LIN {X -0.049,Y -582.708,Z 976.726,A 0.000,B 0.000,C 90.000,E1 346.756} C_DIS
LIN {X 0.095,Y -587.097,Z 976.722,A 0.000,B 0.000,C 90.000,E1 345.936} C_DIS
LIN {X -0.292,Y -591.184,Z 976.718,A 0.000,B 0.000,C 90.000,E1 345.172} C_DIS
LIN {X -0.216,Y -596.425,Z 976.712,A 0.000,B 0.000,C 90.000,E1 344.102} C_DIS
LIN {X 0.105,Y -601.361,Z 976.706,A 0.000,B 0.000,C 90.000,E1 343.015} C_DIS
LIN {X 0.020,Y -604.929,Z 976.701,A 0.000,B 0.000,C 90.000,E1 342.236} C_DIS
LIN {X 0.200,Y -610.324,Z 976.694,A 0.000,B 0.000,C 90.000,E1 340.913} C_DIS
LIN {X 0.140,Y -614.377,Z 976.688,A 0.000,B 0.000,C 90.000,E1 339.880} C_DIS
LIN {X 0.129,Y -618.154,Z 976.683,A 0.000,B 0.000,C 90.000,E1 338.847} C_DIS
LIN {X -0.183,Y -621.682,Z 976.677,A 0.000,B 0.000,C 90.000,E1 337.847} C_DIS
LIN {X 0.136,Y -625.716,Z 976.670,A 0.000,B 0.000,C 90.000,E1 336.538} C_DIS
LIN {X -0.067,Y -628.774,Z 976.664,A 0.000,B 0.000,C 90.000,E1 335.537} C_DIS
LIN {X -0.237,Y -631.659,Z 976.658,A 0.000,B 0.000,C 90.000,E1 334.537} C_DIS
LIN {X -0.099,Y -634.157,Z 976.653,A 0.000,B 0.000,C 90.000,E1 333.512} C_DIS
LIN {X 0.073,Y -636.573,Z 976.647,A 0.000,B 0.000,C 90.000,E1 332.487} C_DIS
LIN {X 0.129,Y -639.825,Z 976.639,A 0.000,B 0.000,C 90.000,E1 330.973} C_DIS
LIN {X -0.192,Y -641.817,Z 976.633,A 0.000,B 0.000,C 90.000,E1 329.999} C_DIS
LIN {X -0.169,Y -643.706,Z 976.628,A 0.000,B 0.000,C 90.000,E1 328.997} C_DIS
LIN {X -0.122,Y -645.317,Z 976.622,A 0.000,B 0.000,C 90.000,E1 327.995} C_DIS
LIN {X -0.061,Y -646.790,Z 976.617,A 0.000,B 0.000,C 90.000,E1 326.993} C_DIS
LIN {X -0.107,Y -648.333,Z 976.610,A 0.000,B 0.000,C 90.000,E1 325.754} C_DIS
LIN {X -0.191,Y -649.344,Z 976.604,A 0.000,B 0.000,C 90.000,E1 324.769} C_DIS
LIN {X 0.098,Y -650.530,Z 976.596,A 0.000,B 0.000,C 90.000,E1 323.256} C_DIS
LIN {X 0.014,Y -651.473,Z 976.588,A 0.000,B 0.000,C 90.000,E1 321.778} C_DIS
LIN {X -0.206,Y -652.064,Z 976.581,A 0.000,B 0.000,C 90.000,E1 320.561} C_DIS
LIN {X 0.057,Y -652.847,Z 976.571,A 0.000,B 0.000,C 90.000,E1 318.809} C_DIS
LIN {X -0.360,Y -654.469,Z 976.558,A 0.000,B 0.000,C 90.000,E1 316.377} C_DIS
LIN {X -0.086,Y -655.453,Z 976.551,A 0.000,B 0.000,C 90.000,E1 315.121} C_DIS
LIN {X 0.068,Y -657.207,Z 976.538,A 0.000,B 0.000,C 90.000,E1 312.894} C_DIS
LIN {X -0.085,Y -658.420,Z 976.530,A 0.000,B 0.000,C 90.000,E1 311.434} C_DIS
LIN {X 0.317,Y -659.253,Z 976.523,A 0.000,B 0.000,C 90.000,E1 310.172} C_DIS
LIN {X -0.186,Y -660.046,Z 976.517,A 0.000,B 0.000,C 90.000,E1 308.991} C_DIS
LIN {X -0.199,Y -660.753,Z 976.508,A 0.000,B 0.000,C 90.000,E1 307.523} C_DIS
LIN {X -0.205,Y -661.096,Z 976.504,A 0.000,B 0.000,C 90.000,E1 306.790} C_DIS
LIN {X 0.408,Y -661.427,Z 976.495,A 0.000,B 0.000,C 90.000,E1 305.025} C_DIS
LIN {X -0.267,Y -661.847,Z 976.485,A 0.000,B 0.000,C 90.000,E1 303.372} C_DIS
LIN {X 0.062,Y -663.392,Z 976.469,A 0.000,B 0.000,C 90.000,E1 300.413} C_DIS
LIN {X 0.159,Y -669.765,Z 976.442,A 0.000,B 0.000,C 90.000,E1 295.540} C_DIS
LIN {X 0.099,Y -671.892,Z 976.435,A 0.000,B 0.000,C 90.000,E1 294.335} C_DIS
LIN {X -0.109,Y -673.447,Z 976.430,A 0.000,B 0.000,C 90.000,E1 293.387} C_DIS
LIN {X -0.030,Y -674.165,Z 976.427,A 0.000,B 0.000,C 90.000,E1 292.898} C_DIS
LIN {X 0.058,Y -674.564,Z 976.425,A 0.000,B 0.000,C 90.000,E1 292.408} C_DIS
LIN {X 0.231,Y -674.612,Z 976.423,A 0.000,B 0.000,C 90.000,E1 292.153} C_DIS
LIN {X -0.302,Y -674.336,Z 976.421,A 0.000,B 0.000,C 90.000,E1 291.716} C_DIS
LIN {X -0.133,Y -673.871,Z 976.419,A 0.000,B 0.000,C 90.000,E1 291.461} C_DIS
LIN {X -0.210,Y -673.270,Z 976.418,A 0.000,B 0.000,C 90.000,E1 291.227} C_DIS
LIN {X -0.044,Y -672.447,Z 976.417,A 0.000,B 0.000,C 90.000,E1 290.972} C_DIS
LIN {X 0.036,Y -671.818,Z 976.416,A 0.000,B 0.000,C 90.000,E1 290.844} C_DIS
LIN {X -0.121,Y -670.864,Z 976.415,A 0.000,B 0.000,C 90.000,E1 290.737} C_DIS
LIN {X 0.152,Y -665.304,Z 976.412,A 0.000,B 0.000,C 90.000,E1 290.194} C_DIS
LIN {X -0.021,Y -657.463,Z 976.409,A 0.000,B 0.000,C 90.000,E1 289.704} C_DIS
LIN {X -0.276,Y -653.001,Z 976.408,A 0.000,B 0.000,C 90.000,E1 289.450} C_DIS
LIN {X 0.214,Y -651.160,Z 976.407,A 0.000,B 0.000,C 90.000,E1 289.214} C_DIS
LIN {X 0.171,Y -651.142,Z 976.407,A 0.000,B 0.000,C 90.000,E1 289.214} C_DIS
LIN {X 0.129,Y -651.087,Z 976.406,A 0.000,B 0.000,C 90.000,E1 289.141} C_DIS
LIN {X -0.058,Y -652.540,Z 976.404,A 0.000,B 0.000,C 90.000,E1 288.725} C_DIS
LIN {X -0.127,Y -656.444,Z 976.400,A 0.000,B 0.000,C 90.000,E1 288.055} C_DIS
LIN {X -0.091,Y -660.813,Z 976.396,A 0.000,B 0.000,C 90.000,E1 287.330} C_DIS
LIN {X -0.246,Y -664.149,Z 976.393,A 0.000,B 0.000,C 90.000,E1 286.732} C_DIS
LIN {X 0.317,Y -667.054,Z 976.390,A 0.000,B 0.000,C 90.000,E1 286.079} C_DIS
LIN {X 0.081,Y -669.685,Z 976.385,A 0.000,B 0.000,C 90.000,E1 285.371} C_DIS
LIN {X -0.060,Y -671.033,Z 976.383,A 0.000,B 0.000,C 90.000,E1 284.898} C_DIS
LIN {X -0.087,Y -672.571,Z 976.379,A 0.000,B 0.000,C 90.000,E1 284.175} C_DIS
LIN {X 0.383,Y -673.703,Z 976.375,A 0.000,B 0.000,C 90.000,E1 283.411} C_DIS
LIN {X 0.060,Y -674.413,Z 976.371,A 0.000,B 0.000,C 90.000,E1 282.715} C_DIS
LIN {X -0.103,Y -674.841,Z 976.367,A 0.000,B 0.000,C 90.000,E1 282.007} C_DIS
LIN {X -0.271,Y -674.764,Z 976.363,A 0.000,B 0.000,C 90.000,E1 281.299} C_DIS
LIN {X 0.148,Y -674.517,Z 976.360,A 0.000,B 0.000,C 90.000,E1 280.782} C_DIS
LIN {X 0.031,Y -673.995,Z 976.357,A 0.000,B 0.000,C 90.000,E1 280.310} C_DIS
LIN {X -0.210,Y -673.266,Z 976.355,A 0.000,B 0.000,C 90.000,E1 279.849} C_DIS
LIN {X 0.322,Y -672.220,Z 976.352,A 0.000,B 0.000,C 90.000,E1 279.321} C_DIS
LIN {X 0.075,Y -670.878,Z 976.349,A 0.000,B 0.000,C 90.000,E1 278.859} C_DIS
LIN {X -0.001,Y -670.147,Z 976.348,A 0.000,B 0.000,C 90.000,E1 278.624} C_DIS
LIN {X -0.259,Y -668.440,Z 976.345,A 0.000,B 0.000,C 90.000,E1 278.163} C_DIS
LIN {X 0.136,Y -666.393,Z 976.343,A 0.000,B 0.000,C 90.000,E1 277.644} C_DIS
LIN {X -0.234,Y -663.311,Z 976.339,A 0.000,B 0.000,C 90.000,E1 277.068} C_DIS
LIN {X 0.104,Y -659.603,Z 976.336,A 0.000,B 0.000,C 90.000,E1 276.429} C_DIS
LIN {X 0.330,Y -655.150,Z 976.332,A 0.000,B 0.000,C 90.000,E1 275.796} C_DIS
LIN {X -0.022,Y -651.196,Z 976.330,A 0.000,B 0.000,C 90.000,E1 275.334} C_DIS
LIN {X 0.191,Y -646.922,Z 976.327,A 0.000,B 0.000,C 90.000,E1 274.821} C_DIS
LIN {X -0.211,Y -642.262,Z 976.324,A 0.000,B 0.000,C 90.000,E1 274.359} C_DIS
LIN {X 0.043,Y -635.920,Z 976.321,A 0.000,B 0.000,C 90.000,E1 273.726} C_DIS
LIN {X -0.093,Y -630.643,Z 976.318,A 0.000,B 0.000,C 90.000,E1 273.269} C_DIS
LIN {X 0.021,Y -625.023,Z 976.316,A 0.000,B 0.000,C 90.000,E1 272.808} C_DIS
LIN {X -0.203,Y -617.622,Z 976.313,A 0.000,B 0.000,C 90.000,E1 272.293} C_DIS
LIN {X -0.222,Y -611.469,Z 976.310,A 0.000,B 0.000,C 90.000,E1 271.892} C_DIS
LIN {X -0.230,Y -603.376,Z 976.308,A 0.000,B 0.000,C 90.000,E1 271.432} C_DIS
LIN {X 0.110,Y -598.334,Z 976.306,A 0.000,B 0.000,C 90.000,E1 271.146} C_DIS
LIN {X -0.088,Y -591.281,Z 976.305,A 0.000,B 0.000,C 90.000,E1 270.859} C_DIS
LIN {X 0.063,Y -584.127,Z 976.303,A 0.000,B 0.000,C 90.000,E1 270.573} C_DIS
LIN {X 0.103,Y -576.473,Z 976.302,A 0.000,B 0.000,C 90.000,E1 270.344} C_DIS
LIN {X -0.244,Y -571.044,Z 976.301,A 0.000,B 0.000,C 90.000,E1 270.229} C_DIS
LIN {X 0.130,Y -564.562,Z 976.300,A 0.000,B 0.000,C 90.000,E1 270.057} C_DIS
LIN {X 0.026,Y -557.390,Z 976.300,A 0.000,B 0.000,C 90.000,E1 270.000} C_DIS
LIN {X -0.024,Y -546.296,Z 976.300,A 0.000,B 0.000,C 90.000,E1 270.000} C_DIS
LIN {X -0.220,Y -544.017,Z 976.300,A 0.000,B 0.000,C 90.000,E1 269.943} C_DIS
LIN {X 0.151,Y -543.248,Z 976.299,A 0.000,B 0.000,C 90.000,E1 269.885} C_DIS
LIN {X 0.108,Y -543.043,Z 976.299,A 0.000,B 0.000,C 90.000,E1 269.885} C_DIS
LIN {X -0.079,Y -542.595,Z 976.298,A 0.000,B 0.000,C 90.000,E1 269.714} C_DIS
LIN {X -0.251,Y -541.922,Z 976.293,A 0.000,B 0.000,C 90.000,E1 268.740} C_DIS
LIN {X -0.045,Y -540.496,Z 976.282,A 0.000,B 0.000,C 90.000,E1 266.731} C_DIS
LIN {X 0.063,Y -539.552,Z 976.274,A 0.000,B 0.000,C 90.000,E1 265.298} C_DIS
LIN {X 0.240,Y -538.503,Z 976.266,A 0.000,B 0.000,C 90.000,E1 263.856} C_DIS
LIN {X -0.127,Y -537.229,Z 976.258,A 0.000,B 0.000,C 90.000,E1 262.470} C_DIS
LIN {X -0.048,Y -536.080,Z 976.252,A 0.000,B 0.000,C 90.000,E1 261.319} C_DIS
LIN {X 0.230,Y -534.668,Z 976.244,A 0.000,B 0.000,C 90.000,E1 259.859} C_DIS
LIN {X -0.087,Y -532.682,Z 976.234,A 0.000,B 0.000,C 90.000,E1 258.173} C_DIS
LIN {X 0.046,Y -531.778,Z 976.229,A 0.000,B 0.000,C 90.000,E1 257.297} C_DIS
LIN {X 0.041,Y -529.264,Z 976.218,A 0.000,B 0.000,C 90.000,E1 255.283} C_DIS
LIN {X -0.204,Y -527.751,Z 976.210,A 0.000,B 0.000,C 90.000,E1 253.866} C_DIS
LIN {X -0.176,Y -525.901,Z 976.201,A 0.000,B 0.000,C 90.000,E1 252.127} C_DIS
LIN {X -0.186,Y -524.098,Z 976.193,A 0.000,B 0.000,C 90.000,E1 250.678} C_DIS
LIN {X 0.102,Y -521.788,Z 976.183,A 0.000,B 0.000,C 90.000,E1 248.901} C_DIS
LIN {X -0.295,Y -519.948,Z 976.175,A 0.000,B 0.000,C 90.000,E1 247.486} C_DIS
LIN {X -0.001,Y -519.209,Z 976.172,A 0.000,B 0.000,C 90.000,E1 246.869} C_DIS
LIN {X 0.099,Y -516.564,Z 976.162,A 0.000,B 0.000,C 90.000,E1 245.101} C_DIS
LIN {X 0.023,Y -514.257,Z 976.154,A 0.000,B 0.000,C 90.000,E1 243.640} C_DIS
LIN {X -0.208,Y -512.415,Z 976.147,A 0.000,B 0.000,C 90.000,E1 242.487} C_DIS
LIN {X 0.112,Y -510.012,Z 976.139,A 0.000,B 0.000,C 90.000,E1 240.973} C_DIS
LIN {X -0.306,Y -507.426,Z 976.131,A 0.000,B 0.000,C 90.000,E1 239.537} C_DIS
LIN {X -0.142,Y -505.116,Z 976.124,A 0.000,B 0.000,C 90.000,E1 238.329} C_DIS
LIN {X -0.134,Y -502.056,Z 976.116,A 0.000,B 0.000,C 90.000,E1 236.834} C_DIS
LIN {X 0.218,Y -499.376,Z 976.109,A 0.000,B 0.000,C 90.000,E1 235.595} C_DIS
LIN {X -0.151,Y -495.265,Z 976.099,A 0.000,B 0.000,C 90.000,E1 233.829} C_DIS
LIN {X 0.227,Y -491.712,Z 976.091,A 0.000,B 0.000,C 90.000,E1 232.271} C_DIS
LIN {X -0.083,Y -488.934,Z 976.084,A 0.000,B 0.000,C 90.000,E1 231.090} C_DIS
LIN {X -0.094,Y -484.579,Z 976.074,A 0.000,B 0.000,C 90.000,E1 229.256} C_DIS
LIN {X 0.057,Y -480.376,Z 976.063,A 0.000,B 0.000,C 90.000,E1 227.391} C_DIS
LIN {X -0.228,Y -476.328,Z 976.053,A 0.000,B 0.000,C 90.000,E1 225.567} C_DIS
LIN {X 0.300,Y -472.927,Z 976.044,A 0.000,B 0.000,C 90.000,E1 223.947} C_DIS
LIN {X 0.192,Y -468.772,Z 976.034,A 0.000,B 0.000,C 90.000,E1 222.081} C_DIS
LIN {X 0.102,Y -466.768,Z 976.029,A 0.000,B 0.000,C 90.000,E1 221.148} C_DIS
LIN {X 0.146,Y -463.236,Z 976.020,A 0.000,B 0.000,C 90.000,E1 219.564} C_DIS
LIN {X -0.049,Y -458.183,Z 976.008,A 0.000,B 0.000,C 90.000,E1 217.363} C_DIS
LIN {X -0.017,Y -453.957,Z 975.997,A 0.000,B 0.000,C 90.000,E1 215.438} C_DIS
LIN {X 0.026,Y -449.715,Z 975.986,A 0.000,B 0.000,C 90.000,E1 213.499} C_DIS
LIN {X 0.035,Y -446.193,Z 975.977,A 0.000,B 0.000,C 90.000,E1 211.878} C_DIS
LIN {X -0.084,Y -443.427,Z 975.970,A 0.000,B 0.000,C 90.000,E1 210.590} C_DIS
LIN {X -0.088,Y -440.629,Z 975.963,A 0.000,B 0.000,C 90.000,E1 209.283} C_DIS
LIN {X 0.139,Y -435.508,Z 975.950,A 0.000,B 0.000,C 90.000,E1 206.950} C_DIS
LIN {X -0.005,Y -433.380,Z 975.944,A 0.000,B 0.000,C 90.000,E1 205.976} C_DIS
LIN {X 0.023,Y -430.297,Z 975.937,A 0.000,B 0.000,C 90.000,E1 204.643} C_DIS
LIN {X -0.074,Y -423.467,Z 975.920,A 0.000,B 0.000,C 90.000,E1 201.642} C_DIS
LIN {X -0.023,Y -418.394,Z 975.907,A 0.000,B 0.000,C 90.000,E1 199.268} C_DIS
LIN {X -0.100,Y -413.003,Z 975.892,A 0.000,B 0.000,C 90.000,E1 196.551} C_DIS
LIN {X -0.036,Y -409.182,Z 975.880,A 0.000,B 0.000,C 90.000,E1 194.481} C_DIS
LIN {X -0.163,Y -405.944,Z 975.871,A 0.000,B 0.000,C 90.000,E1 192.771} C_DIS
LIN {X 0.034,Y -402.616,Z 975.861,A 0.000,B 0.000,C 90.000,E1 191.007} C_DIS
LIN {X 0.014,Y -400.007,Z 975.853,A 0.000,B 0.000,C 90.000,E1 189.613} C_DIS
LIN {X 0.032,Y -393.198,Z 975.832,A 0.000,B 0.000,C 90.000,E1 185.739} C_DIS
LIN {X -0.146,Y -392.071,Z 975.826,A 0.000,B 0.000,C 90.000,E1 184.702} C_DIS
LIN {X 0.105,Y -391.526,Z 975.822,A 0.000,B 0.000,C 90.000,E1 183.955} C_DIS
LIN {X 0.021,Y -391.404,Z 975.820,A 0.000,B 0.000,C 90.000,E1 183.612} C_DIS
LIN {X -0.124,Y -391.727,Z 975.816,A 0.000,B 0.000,C 90.000,E1 182.922} C_DIS
LIN {X 0.185,Y -392.168,Z 975.814,A 0.000,B 0.000,C 90.000,E1 182.522} C_DIS
LIN {X 0.105,Y -392.821,Z 975.812,A 0.000,B 0.000,C 90.000,E1 182.178} C_DIS
LIN {X 0.115,Y -393.673,Z 975.810,A 0.000,B 0.000,C 90.000,E1 181.835} C_DIS
LIN {X 0.047,Y -395.519,Z 975.807,A 0.000,B 0.000,C 90.000,E1 181.318} C_DIS
LIN {X 0.012,Y -397.225,Z 975.805,A 0.000,B 0.000,C 90.000,E1 180.974} C_DIS
LIN {X -0.050,Y -399.256,Z 975.804,A 0.000,B 0.000,C 90.000,E1 180.630} C_DIS
LIN {X -0.136,Y -402.294,Z 975.801,A 0.000,B 0.000,C 90.000,E1 180.229} C_DIS
LIN {X -0.169,Y -405.098,Z 975.799,A 0.000,B 0.000,C 90.000,E1 179.885} C_DIS
LIN {X -0.073,Y -412.702,Z 975.795,A 0.000,B 0.000,C 90.000,E1 179.083} C_DIS
LIN {X 0.071,Y -424.664,Z 975.789,A 0.000,B 0.000,C 90.000,E1 177.936} C_DIS
LIN {X 0.118,Y -436.561,Z 975.782,A 0.000,B 0.000,C 90.000,E1 176.788} C_DIS
LIN {X -0.066,Y -440.929,Z 975.780,A 0.000,B 0.000,C 90.000,E1 176.388} C_DIS
LIN {X -0.137,Y -449.606,Z 975.775,A 0.000,B 0.000,C 90.000,E1 175.527} C_DIS
LIN {X 0.185,Y -460.939,Z 975.769,A 0.000,B 0.000,C 90.000,E1 174.318} C_DIS
LIN {X 0.115,Y -470.380,Z 975.763,A 0.000,B 0.000,C 90.000,E1 173.280} C_DIS
LIN {X 0.092,Y -478.131,Z 975.758,A 0.000,B 0.000,C 90.000,E1 172.356} C_DIS
LIN {X 0.048,Y -485.586,Z 975.753,A 0.000,B 0.000,C 90.000,E1 171.432} C_DIS
LIN {X 0.059,Y -494.990,Z 975.746,A 0.000,B 0.000,C 90.000,E1 170.208} C_DIS
LIN {X -0.040,Y -502.686,Z 975.740,A 0.000,B 0.000,C 90.000,E1 169.162} C_DIS
LIN {X 0.231,Y -510.899,Z 975.733,A 0.000,B 0.000,C 90.000,E1 167.937} C_DIS
LIN {X 0.250,Y -520.550,Z 975.725,A 0.000,B 0.000,C 90.000,E1 166.464} C_DIS
LIN {X 0.063,Y -524.967,Z 975.721,A 0.000,B 0.000,C 90.000,E1 165.755} C_DIS
LIN {X -0.066,Y -531.342,Z 975.715,A 0.000,B 0.000,C 90.000,E1 164.755} C_DIS
LIN {X -0.133,Y -538.234,Z 975.709,A 0.000,B 0.000,C 90.000,E1 163.614} C_DIS
LIN {X -0.257,Y -544.932,Z 975.703,A 0.000,B 0.000,C 90.000,E1 162.489} C_DIS
LIN {X 0.134,Y -553.029,Z 975.695,A 0.000,B 0.000,C 90.000,E1 161.040} C_DIS
LIN {X -0.068,Y -560.210,Z 975.688,A 0.000,B 0.000,C 90.000,E1 159.806} C_DIS
LIN {X 0.150,Y -564.674,Z 975.683,A 0.000,B 0.000,C 90.000,E1 158.954} C_DIS
LIN {X 0.229,Y -570.421,Z 975.677,A 0.000,B 0.000,C 90.000,E1 157.847} C_DIS
LIN {X 0.019,Y -574.548,Z 975.673,A 0.000,B 0.000,C 90.000,E1 157.050} C_DIS
LIN {X 0.149,Y -577.818,Z 975.669,A 0.000,B 0.000,C 90.000,E1 156.357} C_DIS
LIN {X 0.175,Y -582.234,Z 975.664,A 0.000,B 0.000,C 90.000,E1 155.409} C_DIS
LIN {X 0.253,Y -586.241,Z 975.658,A 0.000,B 0.000,C 90.000,E1 154.460} C_DIS
LIN {X -0.099,Y -589.497,Z 975.654,A 0.000,B 0.000,C 90.000,E1 153.691} C_DIS
LIN {X 0.007,Y -593.406,Z 975.648,A 0.000,B 0.000,C 90.000,E1 152.615} C_DIS
LIN {X -0.088,Y -596.866,Z 975.642,A 0.000,B 0.000,C 90.000,E1 151.563} C_DIS
LIN {X -0.208,Y -600.991,Z 975.635,A 0.000,B 0.000,C 90.000,E1 150.255} C_DIS
LIN {X 0.044,Y -605.049,Z 975.627,A 0.000,B 0.000,C 90.000,E1 148.918} C_DIS
LIN {X 0.104,Y -608.260,Z 975.622,A 0.000,B 0.000,C 90.000,E1 147.867} C_DIS
LIN {X 0.012,Y -611.516,Z 975.616,A 0.000,B 0.000,C 90.000,E1 146.834} C_DIS
LIN {X 0.009,Y -617.095,Z 975.606,A 0.000,B 0.000,C 90.000,E1 145.022} C_DIS
LIN {X -0.192,Y -621.794,Z 975.597,A 0.000,B 0.000,C 90.000,E1 143.497} C_DIS
LIN {X -0.056,Y -626.495,Z 975.589,A 0.000,B 0.000,C 90.000,E1 141.949} C_DIS
LIN {X -0.209,Y -631.159,Z 975.580,A 0.000,B 0.000,C 90.000,E1 140.436} C_DIS
LIN {X -0.367,Y -635.644,Z 975.572,A 0.000,B 0.000,C 90.000,E1 138.933} C_DIS
LIN {X 0.195,Y -642.570,Z 975.559,A 0.000,B 0.000,C 90.000,E1 136.620} C_DIS
LIN {X -0.247,Y -647.308,Z 975.551,A 0.000,B 0.000,C 90.000,E1 135.162} C_DIS
LIN {X -0.304,Y -655.718,Z 975.537,A 0.000,B 0.000,C 90.000,E1 132.690} C_DIS
LIN {X -0.057,Y -664.670,Z 975.523,A 0.000,B 0.000,C 90.000,E1 130.216} C_DIS
LIN {X -0.041,Y -668.186,Z 975.518,A 0.000,B 0.000,C 90.000,E1 129.241} C_DIS
LIN {X -0.299,Y -673.284,Z 975.510,A 0.000,B 0.000,C 90.000,E1 127.810} C_DIS
LIN {X -0.047,Y -677.105,Z 975.503,A 0.000,B 0.000,C 90.000,E1 126.583} C_DIS
LIN {X -0.133,Y -680.780,Z 975.497,A 0.000,B 0.000,C 90.000,E1 125.391} C_DIS
LIN {X 0.222,Y -683.642,Z 975.491,A 0.000,B 0.000,C 90.000,E1 124.405} C_DIS
LIN {X -0.143,Y -686.979,Z 975.485,A 0.000,B 0.000,C 90.000,E1 123.245} C_DIS
LIN {X 0.131,Y -690.701,Z 975.477,A 0.000,B 0.000,C 90.000,E1 121.799} C_DIS
LIN {X -0.134,Y -693.018,Z 975.471,A 0.000,B 0.000,C 90.000,E1 120.875} C_DIS
LIN {X 0.340,Y -694.597,Z 975.468,A 0.000,B 0.000,C 90.000,E1 120.129} C_DIS
LIN {X -0.126,Y -695.992,Z 975.464,A 0.000,B 0.000,C 90.000,E1 119.461} C_DIS
LIN {X 0.283,Y -697.433,Z 975.458,A 0.000,B 0.000,C 90.000,E1 118.487} C_DIS
LIN {X 0.037,Y -698.610,Z 975.452,A 0.000,B 0.000,C 90.000,E1 117.334} C_DIS
LIN {X 0.215,Y -699.315,Z 975.448,A 0.000,B 0.000,C 90.000,E1 116.616} C_DIS
LIN {X -0.003,Y -700.165,Z 975.442,A 0.000,B 0.000,C 90.000,E1 115.463} C_DIS
LIN {X -0.122,Y -700.448,Z 975.438,A 0.000,B 0.000,C 90.000,E1 114.771} C_DIS
LIN {X 0.130,Y -700.507,Z 975.435,A 0.000,B 0.000,C 90.000,E1 114.283} C_DIS
LIN {X 0.032,Y -700.124,Z 975.432,A 0.000,B 0.000,C 90.000,E1 113.823} C_DIS
LIN {X 0.019,Y -699.837,Z 975.431,A 0.000,B 0.000,C 90.000,E1 113.590} C_DIS
LIN {X -0.090,Y -698.362,Z 975.429,A 0.000,B 0.000,C 90.000,E1 113.131} C_DIS
LIN {X -0.101,Y -697.334,Z 975.427,A 0.000,B 0.000,C 90.000,E1 112.898} C_DIS
LIN {X 0.156,Y -695.329,Z 975.426,A 0.000,B 0.000,C 90.000,E1 112.642} C_DIS
LIN {X 0.262,Y -691.942,Z 975.424,A 0.000,B 0.000,C 90.000,E1 112.280} C_DIS
LIN {X -0.257,Y -690.182,Z 975.423,A 0.000,B 0.000,C 90.000,E1 112.206} C_DIS
LIN {X 0.245,Y -685.451,Z 975.422,A 0.000,B 0.000,C 90.000,E1 111.972} C_DIS
LIN {X 0.347,Y -683.290,Z 975.422,A 0.000,B 0.000,C 90.000,E1 111.897} C_DIS
LIN {X -0.209,Y -675.865,Z 975.421,A 0.000,B 0.000,C 90.000,E1 111.770} C_DIS
LIN {X 0.240,Y -674.512,Z 975.421,A 0.000,B 0.000,C 90.000,E1 111.716} C_DIS
LIN {X 0.175,Y -672.657,Z 975.421,A 0.000,B 0.000,C 90.000,E1 111.716} C_DIS
LIN {X 0.104,Y -626.026,Z 975.421,A 0.000,B 0.000,C 90.000,E1 111.716} C_DIS
LIN {X -0.147,Y -621.534,Z 975.420,A 0.000,B 0.000,C 90.000,E1 111.663} C_DIS
LIN {X -0.200,Y -615.743,Z 975.420,A 0.000,B 0.000,C 90.000,E1 111.535} C_DIS
LIN {X -0.047,Y -610.298,Z 975.419,A 0.000,B 0.000,C 90.000,E1 111.354} C_DIS
LIN {X -0.253,Y -603.607,Z 975.417,A 0.000,B 0.000,C 90.000,E1 111.099} C_DIS
LIN {X 0.138,Y -597.489,Z 975.415,A 0.000,B 0.000,C 90.000,E1 110.737} C_DIS
LIN {X -0.152,Y -590.496,Z 975.413,A 0.000,B 0.000,C 90.000,E1 110.301} C_DIS
LIN {X 0.287,Y -578.355,Z 975.408,A 0.000,B 0.000,C 90.000,E1 109.322} C_DIS
LIN {X -0.163,Y -573.848,Z 975.406,A 0.000,B 0.000,C 90.000,E1 109.033} C_DIS
LIN {X 0.152,Y -567.242,Z 975.403,A 0.000,B 0.000,C 90.000,E1 108.598} C_DIS
LIN {X 0.208,Y -552.115,Z 975.399,A 0.000,B 0.000,C 90.000,E1 107.819} C_DIS
LIN {X 0.101,Y -549.945,Z 975.398,A 0.000,B 0.000,C 90.000,E1 107.638} C_DIS
LIN {X 0.064,Y -549.916,Z 975.398,A 0.000,B 0.000,C 90.000,E1 107.638} C_DIS
LIN {X -0.275,Y -549.445,Z 975.397,A 0.000,B 0.000,C 90.000,E1 107.402} C_DIS
LIN {X -0.059,Y -549.569,Z 975.393,A 0.000,B 0.000,C 90.000,E1 106.677} C_DIS
LIN {X -0.107,Y -550.406,Z 975.382,A 0.000,B 0.000,C 90.000,E1 104.717} C_DIS
LIN {X -0.266,Y -551.503,Z 975.371,A 0.000,B 0.000,C 90.000,E1 102.771} C_DIS
LIN {X -0.152,Y -553.940,Z 975.355,A 0.000,B 0.000,C 90.000,E1 99.962} C_DIS
LIN {X -0.041,Y -555.670,Z 975.346,A 0.000,B 0.000,C 90.000,E1 98.276} C_DIS
LIN {X -0.046,Y -557.231,Z 975.337,A 0.000,B 0.000,C 90.000,E1 96.606} C_DIS
LIN {X -0.083,Y -558.317,Z 975.329,A 0.000,B 0.000,C 90.000,E1 95.220} C_DIS
LIN {X -0.160,Y -559.230,Z 975.321,A 0.000,B 0.000,C 90.000,E1 93.841} C_DIS
LIN {X 0.126,Y -559.732,Z 975.317,A 0.000,B 0.000,C 90.000,E1 92.980} C_DIS
LIN {X 0.037,Y -560.476,Z 975.309,A 0.000,B 0.000,C 90.000,E1 91.604} C_DIS
LIN {X 0.045,Y -561.266,Z 975.300,A 0.000,B 0.000,C 90.000,E1 89.943} C_DIS
LIN {X -0.028,Y -561.686,Z 975.292,A 0.000,B 0.000,C 90.000,E1 88.568} C_DIS
LIN {X 0.012,Y -562.097,Z 975.283,A 0.000,B 0.000,C 90.000,E1 86.906} C_DIS
LIN {X -0.004,Y -562.312,Z 975.275,A 0.000,B 0.000,C 90.000,E1 85.527} C_DIS
LIN {X 0.219,Y -562.559,Z 975.264,A 0.000,B 0.000,C 90.000,E1 83.571} C_DIS
LIN {X 0.096,Y -562.955,Z 975.252,A 0.000,B 0.000,C 90.000,E1 81.376} C_DIS
LIN {X 0.004,Y -563.655,Z 975.241,A 0.000,B 0.000,C 90.000,E1 79.454} C_DIS
LIN {X 0.215,Y -564.684,Z 975.229,A 0.000,B 0.000,C 90.000,E1 77.229} C_DIS
LIN {X 0.031,Y -566.117,Z 975.217,A 0.000,B 0.000,C 90.000,E1 75.046} C_DIS
LIN {X -0.142,Y -567.444,Z 975.206,A 0.000,B 0.000,C 90.000,E1 73.142} C_DIS
LIN {X -0.081,Y -568.345,Z 975.199,A 0.000,B 0.000,C 90.000,E1 71.764} C_DIS
LIN {X -0.019,Y -569.347,Z 975.190,A 0.000,B 0.000,C 90.000,E1 70.115} C_DIS
LIN {X 0.253,Y -570.077,Z 975.182,A 0.000,B 0.000,C 90.000,E1 68.720} C_DIS
LIN {X -0.147,Y -570.536,Z 975.176,A 0.000,B 0.000,C 90.000,E1 67.667} C_DIS
LIN {X -0.188,Y -571.056,Z 975.168,A 0.000,B 0.000,C 90.000,E1 66.305} C_DIS
LIN {X -0.164,Y -571.570,Z 975.159,A 0.000,B 0.000,C 90.000,E1 64.665} C_DIS
LIN {X 0.287,Y -571.934,Z 975.152,A 0.000,B 0.000,C 90.000,E1 63.256} C_DIS
LIN {X 0.237,Y -572.190,Z 975.144,A 0.000,B 0.000,C 90.000,E1 61.897} C_DIS
LIN {X 0.020,Y -572.367,Z 975.135,A 0.000,B 0.000,C 90.000,E1 60.284} C_DIS
LIN {X -0.125,Y -572.538,Z 975.126,A 0.000,B 0.000,C 90.000,E1 58.663} C_DIS
LIN {X -0.255,Y -572.717,Z 975.117,A 0.000,B 0.000,C 90.000,E1 57.041} C_DIS
LIN {X -0.210,Y -572.707,Z 975.109,A 0.000,B 0.000,C 90.000,E1 55.674} C_DIS
LIN {X -0.123,Y -572.624,Z 975.105,A 0.000,B 0.000,C 90.000,E1 54.848} C_DIS
LIN {X -0.030,Y -572.276,Z 975.099,A 0.000,B 0.000,C 90.000,E1 53.749} C_DIS
LIN {X 0.047,Y -571.928,Z 975.094,A 0.000,B 0.000,C 90.000,E1 52.924} C_DIS
LIN {X 0.277,Y -571.193,Z 975.087,A 0.000,B 0.000,C 90.000,E1 51.537} C_DIS
LIN {X 0.231,Y -570.598,Z 975.082,A 0.000,B 0.000,C 90.000,E1 50.723} C_DIS
LIN {X -0.129,Y -569.538,Z 975.076,A 0.000,B 0.000,C 90.000,E1 49.666} C_DIS
LIN {X -0.074,Y -568.281,Z 975.070,A 0.000,B 0.000,C 90.000,E1 48.566} C_DIS
LIN {X 0.108,Y -567.601,Z 975.067,A 0.000,B 0.000,C 90.000,E1 48.000} C_DIS
LIN {X 0.084,Y -565.863,Z 975.061,A 0.000,B 0.000,C 90.000,E1 46.905} C_DIS
LIN {X 0.352,Y -564.365,Z 975.056,A 0.000,B 0.000,C 90.000,E1 46.053} C_DIS
LIN {X -0.126,Y -562.088,Z 975.050,A 0.000,B 0.000,C 90.000,E1 45.000} C_DIS
LIN {X 0.159,Y -559.262,Z 975.044,A 0.000,B 0.000,C 90.000,E1 43.866} C_DIS
LIN {X -0.054,Y -556.893,Z 975.039,A 0.000,B 0.000,C 90.000,E1 43.056} C_DIS
LIN {X 0.112,Y -554.266,Z 975.035,A 0.000,B 0.000,C 90.000,E1 42.204} C_DIS
LIN {X -0.116,Y -551.191,Z 975.030,A 0.000,B 0.000,C 90.000,E1 41.391} C_DIS
LIN {X -0.009,Y -547.789,Z 975.025,A 0.000,B 0.000,C 90.000,E1 40.539} C_DIS
LIN {X -0.143,Y -544.729,Z 975.021,A 0.000,B 0.000,C 90.000,E1 39.850} C_DIS
LIN {X -0.075,Y -542.061,Z 975.018,A 0.000,B 0.000,C 90.000,E1 39.277} C_DIS
LIN {X 0.136,Y -539.950,Z 975.016,A 0.000,B 0.000,C 90.000,E1 38.830} C_DIS
LIN {X -0.234,Y -533.895,Z 975.010,A 0.000,B 0.000,C 90.000,E1 37.729} C_DIS
LIN {X -0.266,Y -527.366,Z 975.003,A 0.000,B 0.000,C 90.000,E1 36.583} C_DIS
LIN {X 0.203,Y -521.301,Z 974.997,A 0.000,B 0.000,C 90.000,E1 35.518} C_DIS
LIN {X -0.136,Y -514.752,Z 974.992,A 0.000,B 0.000,C 90.000,E1 34.532} C_DIS
LIN {X -0.045,Y -509.671,Z 974.988,A 0.000,B 0.000,C 90.000,E1 33.785} C_DIS
LIN {X 0.223,Y -503.070,Z 974.983,A 0.000,B 0.000,C 90.000,E1 32.880} C_DIS
LIN {X -0.087,Y -499.490,Z 974.980,A 0.000,B 0.000,C 90.000,E1 32.467} C_DIS
LIN {X -0.126,Y -493.015,Z 974.976,A 0.000,B 0.000,C 90.000,E1 31.720} C_DIS
LIN {X 0.081,Y -486.240,Z 974.972,A 0.000,B 0.000,C 90.000,E1 30.954} C_DIS
LIN {X -0.181,Y -476.280,Z 974.967,A 0.000,B 0.000,C 90.000,E1 30.001} C_DIS
LIN {X 0.110,Y -469.132,Z 974.963,A 0.000,B 0.000,C 90.000,E1 29.283} C_DIS
LIN {X -0.010,Y -458.843,Z 974.958,A 0.000,B 0.000,C 90.000,E1 28.359} C_DIS
LIN {X -0.048,Y -449.667,Z 974.953,A 0.000,B 0.000,C 90.000,E1 27.564} C_DIS
LIN {X -0.005,Y -428.305,Z 974.943,A 0.000,B 0.000,C 90.000,E1 25.720} C_DIS
LIN {X 0.030,Y -413.569,Z 974.935,A 0.000,B 0.000,C 90.000,E1 24.335} C_DIS
LIN {X 0.057,Y -403.735,Z 974.930,A 0.000,B 0.000,C 90.000,E1 23.334} C_DIS
LIN {X -0.171,Y -396.868,Z 974.925,A 0.000,B 0.000,C 90.000,E1 22.589} C_DIS
LIN {X -0.155,Y -393.836,Z 974.923,A 0.000,B 0.000,C 90.000,E1 22.153} C_DIS
LIN {X -0.190,Y -391.547,Z 974.921,A 0.000,B 0.000,C 90.000,E1 21.716} C_DIS
LIN {X 0.076,Y -391.215,Z 974.920,A 0.000,B 0.000,C 90.000,E1 21.589} C_DIS
LIN {X 0.122,Y -390.373,Z 974.918,A 0.000,B 0.000,C 90.000,E1 21.227} C_DIS
LIN {X 0.144,Y -390.132,Z 974.917,A 0.000,B 0.000,C 90.000,E1 21.046} C_DIS
LIN {X -0.157,Y -389.856,Z 974.914,A 0.000,B 0.000,C 90.000,E1 20.556} C_DIS
LIN {X 0.058,Y -390.035,Z 974.910,A 0.000,B 0.000,C 90.000,E1 19.812} C_DIS
LIN {X 0.072,Y -394.488,Z 974.885,A 0.000,B 0.000,C 90.000,E1 15.190} C_DIS
LIN {X 0.150,Y -398.153,Z 974.869,A 0.000,B 0.000,C 90.000,E1 12.355} C_DIS
LIN {X 0.087,Y -404.277,Z 974.847,A 0.000,B 0.000,C 90.000,E1 8.511} C_DIS
LIN {X 0.071,Y -410.146,Z 974.830,A 0.000,B 0.000,C 90.000,E1 5.391} C_DIS
LIN {X 0.108,Y -415.225,Z 974.817,A 0.000,B 0.000,C 90.000,E1 2.980} C_DIS
LIN {X -0.164,Y -420.827,Z 974.803,A 0.000,B 0.000,C 90.000,E1 0.630} C_DIS
LIN {X 0.000,Y -422.821,Z 974.800,A 0.000,B 0.000,C 90.000,E1 360.000} C_DIS
LIN {X 0.135,Y -425.410,Z 974.797,A 0.000,B 0.000,C 90.000,E1 359.484} C_DIS
LIN {X 0.185,Y -427.893,Z 974.795,A 0.000,B 0.000,C 90.000,E1 359.141} C_DIS
LIN {X 0.021,Y -429.986,Z 974.794,A 0.000,B 0.000,C 90.000,E1 358.912} C_DIS
LIN {X -0.063,Y -433.565,Z 974.792,A 0.000,B 0.000,C 90.000,E1 358.625} C_DIS
LIN {X -0.163,Y -435.456,Z 974.792,A 0.000,B 0.000,C 90.000,E1 358.511} C_DIS
LIN {X 0.123,Y -454.709,Z 974.786,A 0.000,B 0.000,C 90.000,E1 357.421} C_DIS
LIN {X -0.067,Y -469.854,Z 974.781,A 0.000,B 0.000,C 90.000,E1 356.617} C_DIS
LIN {X -0.072,Y -478.335,Z 974.779,A 0.000,B 0.000,C 90.000,E1 356.159} C_DIS
LIN {X -0.096,Y -491.329,Z 974.774,A 0.000,B 0.000,C 90.000,E1 355.412} C_DIS
LIN {X -0.101,Y -501.296,Z 974.771,A 0.000,B 0.000,C 90.000,E1 354.837} C_DIS
LIN {X -0.202,Y -510.939,Z 974.768,A 0.000,B 0.000,C 90.000,E1 354.261} C_DIS
LIN {X -0.052,Y -520.205,Z 974.765,A 0.000,B 0.000,C 90.000,E1 353.628} C_DIS
LIN {X -0.268,Y -527.938,Z 974.762,A 0.000,B 0.000,C 90.000,E1 353.109} C_DIS
LIN {X -0.117,Y -535.291,Z 974.758,A 0.000,B 0.000,C 90.000,E1 352.527} C_DIS
LIN {X 0.189,Y -542.337,Z 974.755,A 0.000,B 0.000,C 90.000,E1 351.894} C_DIS
LIN {X 0.174,Y -549.039,Z 974.752,A 0.000,B 0.000,C 90.000,E1 351.254} C_DIS
LIN {X 0.054,Y -554.220,Z 974.749,A 0.000,B 0.000,C 90.000,E1 350.735} C_DIS
LIN {X -0.126,Y -559.005,Z 974.746,A 0.000,B 0.000,C 90.000,E1 350.208} C_DIS
LIN {X 0.146,Y -565.207,Z 974.741,A 0.000,B 0.000,C 90.000,E1 349.398} C_DIS
LIN {X -0.073,Y -569.266,Z 974.738,A 0.000,B 0.000,C 90.000,E1 348.870} C_DIS
LIN {X 0.299,Y -573.075,Z 974.735,A 0.000,B 0.000,C 90.000,E1 348.285} C_DIS
LIN {X -0.102,Y -577.363,Z 974.731,A 0.000,B 0.000,C 90.000,E1 347.645} C_DIS
LIN {X -0.120,Y -582.918,Z 974.726,A 0.000,B 0.000,C 90.000,E1 346.700} C_DIS
LIN {X 0.024,Y -587.302,Z 974.722,A 0.000,B 0.000,C 90.000,E1 345.880} C_DIS
LIN {X -0.212,Y -591.432,Z 974.717,A 0.000,B 0.000,C 90.000,E1 345.102} C_DIS
LIN {X -0.124,Y -596.679,Z 974.711,A 0.000,B 0.000,C 90.000,E1 344.031} C_DIS
LIN {X 0.090,Y -601.039,Z 974.706,A 0.000,B 0.000,C 90.000,E1 343.087} C_DIS
LIN {X -0.052,Y -605.189,Z 974.701,A 0.000,B 0.000,C 90.000,E1 342.181} C_DIS
LIN {X 0.127,Y -610.591,Z 974.694,A 0.000,B 0.000,C 90.000,E1 340.859} C_DIS
LIN {X 0.326,Y -613.712,Z 974.689,A 0.000,B 0.000,C 90.000,E1 340.061} C_DIS
LIN {X -0.267,Y -617.569,Z 974.684,A 0.000,B 0.000,C 90.000,E1 339.082} C_DIS
LIN {X -0.257,Y -621.991,Z 974.677,A 0.000,B 0.000,C 90.000,E1 337.794} C_DIS
LIN {X 0.058,Y -625.265,Z 974.671,A 0.000,B 0.000,C 90.000,E1 336.741} C_DIS
LIN {X -0.158,Y -628.399,Z 974.665,A 0.000,B 0.000,C 90.000,E1 335.741} C_DIS
LIN {X -0.069,Y -631.304,Z 974.660,A 0.000,B 0.000,C 90.000,E1 334.717} C_DIS
LIN {X 0.030,Y -633.310,Z 974.655,A 0.000,B 0.000,C 90.000,E1 333.948} C_DIS
LIN {X 0.292,Y -636.971,Z 974.647,A 0.000,B 0.000,C 90.000,E1 332.410} C_DIS
LIN {X 0.053,Y -640.240,Z 974.639,A 0.000,B 0.000,C 90.000,E1 330.923} C_DIS
LIN {X 0.053,Y -642.241,Z 974.633,A 0.000,B 0.000,C 90.000,E1 329.921} C_DIS
LIN {X -0.246,Y -644.139,Z 974.627,A 0.000,B 0.000,C 90.000,E1 328.948} C_DIS
LIN {X -0.265,Y -645.360,Z 974.623,A 0.000,B 0.000,C 90.000,E1 328.201} C_DIS
LIN {X 0.215,Y -647.202,Z 974.616,A 0.000,B 0.000,C 90.000,E1 326.914} C_DIS
LIN {X 0.181,Y -648.733,Z 974.609,A 0.000,B 0.000,C 90.000,E1 325.674} C_DIS
LIN {X 0.105,Y -649.743,Z 974.604,A 0.000,B 0.000,C 90.000,E1 324.689} C_DIS
LIN {X -0.038,Y -650.781,Z 974.597,A 0.000,B 0.000,C 90.000,E1 323.463} C_DIS
LIN {X 0.360,Y -651.626,Z 974.590,A 0.000,B 0.000,C 90.000,E1 322.190} C_DIS
LIN {X 0.243,Y -652.290,Z 974.583,A 0.000,B 0.000,C 90.000,E1 320.964} C_DIS
LIN {X 0.010,Y -653.079,Z 974.574,A 0.000,B 0.000,C 90.000,E1 319.256} C_DIS
LIN {X 0.002,Y -654.983,Z 974.557,A 0.000,B 0.000,C 90.000,E1 316.296} C_DIS
LIN {X -0.179,Y -655.937,Z 974.550,A 0.000,B 0.000,C 90.000,E1 315.081} C_DIS
LIN {X 0.038,Y -657.559,Z 974.539,A 0.000,B 0.000,C 90.000,E1 313.095} C_DIS
LIN {X -0.124,Y -658.969,Z 974.530,A 0.000,B 0.000,C 90.000,E1 311.391} C_DIS
LIN {X -0.207,Y -659.807,Z 974.523,A 0.000,B 0.000,C 90.000,E1 310.172} C_DIS
LIN {X 0.227,Y -660.599,Z 974.516,A 0.000,B 0.000,C 90.000,E1 308.910} C_DIS
LIN {X 0.223,Y -661.330,Z 974.508,A 0.000,B 0.000,C 90.000,E1 307.443} C_DIS
LIN {X -0.174,Y -661.634,Z 974.504,A 0.000,B 0.000,C 90.000,E1 306.744} C_DIS
LIN {X 0.358,Y -661.959,Z 974.496,A 0.000,B 0.000,C 90.000,E1 305.231} C_DIS
LIN {X -0.306,Y -662.391,Z 974.486,A 0.000,B 0.000,C 90.000,E1 303.579} C_DIS
LIN {X -0.071,Y -664.876,Z 974.463,A 0.000,B 0.000,C 90.000,E1 299.411} C_DIS
LIN {X -0.129,Y -670.017,Z 974.443,A 0.000,B 0.000,C 90.000,E1 295.771} C_DIS
LIN {X -0.307,Y -672.537,Z 974.435,A 0.000,B 0.000,C 90.000,E1 294.335} C_DIS
LIN {X 0.111,Y -674.133,Z 974.430,A 0.000,B 0.000,C 90.000,E1 293.334} C_DIS
LIN {X -0.424,Y -674.865,Z 974.427,A 0.000,B 0.000,C 90.000,E1 292.898} C_DIS
LIN {X -0.075,Y -675.208,Z 974.424,A 0.000,B 0.000,C 90.000,E1 292.386} C_DIS
LIN {X -0.157,Y -675.244,Z 974.423,A 0.000,B 0.000,C 90.000,E1 292.153} C_DIS
LIN {X -0.059,Y -674.876,Z 974.420,A 0.000,B 0.000,C 90.000,E1 291.663} C_DIS
LIN {X 0.113,Y -674.378,Z 974.419,A 0.000,B 0.000,C 90.000,E1 291.408} C_DIS
LIN {X 0.207,Y -672.741,Z 974.416,A 0.000,B 0.000,C 90.000,E1 290.918} C_DIS
LIN {X 0.288,Y -672.065,Z 974.416,A 0.000,B 0.000,C 90.000,E1 290.791} C_DIS
LIN {X 0.132,Y -671.047,Z 974.415,A 0.000,B 0.000,C 90.000,E1 290.684} C_DIS
LIN {X 0.287,Y -668.169,Z 974.414,A 0.000,B 0.000,C 90.000,E1 290.429} C_DIS
LIN {X -0.141,Y -665.907,Z 974.412,A 0.000,B 0.000,C 90.000,E1 290.248} C_DIS
LIN {X 0.064,Y -662.387,Z 974.411,A 0.000,B 0.000,C 90.000,E1 289.993} C_DIS
LIN {X 0.045,Y -653.657,Z 974.408,A 0.000,B 0.000,C 90.000,E1 289.450} C_DIS
LIN {X 0.284,Y -652.209,Z 974.407,A 0.000,B 0.000,C 90.000,E1 289.268} C_DIS
LIN {X 0.250,Y -652.186,Z 974.407,A 0.000,B 0.000,C 90.000,E1 289.268} C_DIS
LIN {X -0.015,Y -652.108,Z 974.406,A 0.000,B 0.000,C 90.000,E1 289.141} C_DIS
LIN {X -0.111,Y -653.396,Z 974.404,A 0.000,B 0.000,C 90.000,E1 288.779} C_DIS
LIN {X -0.243,Y -654.685,Z 974.403,A 0.000,B 0.000,C 90.000,E1 288.544} C_DIS
LIN {X 0.163,Y -661.336,Z 974.397,A 0.000,B 0.000,C 90.000,E1 287.402} C_DIS
LIN {X 0.017,Y -664.697,Z 974.393,A 0.000,B 0.000,C 90.000,E1 286.804} C_DIS
LIN {X -0.055,Y -668.154,Z 974.389,A 0.000,B 0.000,C 90.000,E1 286.079} C_DIS
LIN {X -0.281,Y -670.708,Z 974.385,A 0.000,B 0.000,C 90.000,E1 285.371} C_DIS
LIN {X -0.244,Y -672.024,Z 974.383,A 0.000,B 0.000,C 90.000,E1 284.883} C_DIS
LIN {X 0.217,Y -673.532,Z 974.379,A 0.000,B 0.000,C 90.000,E1 284.120} C_DIS
LIN {X 0.101,Y -674.363,Z 974.376,A 0.000,B 0.000,C 90.000,E1 283.647} C_DIS
LIN {X -0.066,Y -675.173,Z 974.372,A 0.000,B 0.000,C 90.000,E1 282.939} C_DIS
LIN {X -0.373,Y -675.671,Z 974.368,A 0.000,B 0.000,C 90.000,E1 282.243} C_DIS
LIN {X 0.236,Y -675.812,Z 974.367,A 0.000,B 0.000,C 90.000,E1 281.951} C_DIS
LIN {X 0.080,Y -675.746,Z 974.363,A 0.000,B 0.000,C 90.000,E1 281.243} C_DIS
LIN {X -0.156,Y -675.492,Z 974.360,A 0.000,B 0.000,C 90.000,E1 280.782} C_DIS
LIN {X -0.267,Y -674.972,Z 974.357,A 0.000,B 0.000,C 90.000,E1 280.310} C_DIS
LIN {X 0.162,Y -674.239,Z 974.355,A 0.000,B 0.000,C 90.000,E1 279.792} C_DIS
LIN {X 0.038,Y -673.166,Z 974.352,A 0.000,B 0.000,C 90.000,E1 279.321} C_DIS
LIN {X -0.204,Y -671.815,Z 974.349,A 0.000,B 0.000,C 90.000,E1 278.859} C_DIS
LIN {X 0.213,Y -670.231,Z 974.346,A 0.000,B 0.000,C 90.000,E1 278.341} C_DIS
LIN {X 0.135,Y -669.395,Z 974.345,A 0.000,B 0.000,C 90.000,E1 278.106} C_DIS
LIN {X -0.126,Y -667.318,Z 974.342,A 0.000,B 0.000,C 90.000,E1 277.644} C_DIS
LIN {X 0.172,Y -664.252,Z 974.339,A 0.000,B 0.000,C 90.000,E1 277.011} C_DIS
LIN {X -0.139,Y -660.566,Z 974.336,A 0.000,B 0.000,C 90.000,E1 276.429} C_DIS
LIN {X 0.197,Y -657.098,Z 974.333,A 0.000,B 0.000,C 90.000,E1 275.910} C_DIS
LIN {X -0.249,Y -652.207,Z 974.330,A 0.000,B 0.000,C 90.000,E1 275.334} C_DIS
LIN {X -0.028,Y -647.982,Z 974.327,A 0.000,B 0.000,C 90.000,E1 274.821} C_DIS
LIN {X 0.221,Y -643.370,Z 974.324,A 0.000,B 0.000,C 90.000,E1 274.302} C_DIS
LIN {X -0.158,Y -637.097,Z 974.321,A 0.000,B 0.000,C 90.000,E1 273.726} C_DIS
LIN {X -0.324,Y -631.846,Z 974.318,A 0.000,B 0.000,C 90.000,E1 273.269} C_DIS
LIN {X -0.221,Y -624.768,Z 974.315,A 0.000,B 0.000,C 90.000,E1 272.694} C_DIS
LIN {X 0.261,Y -617.397,Z 974.312,A 0.000,B 0.000,C 90.000,E1 272.121} C_DIS
LIN {X 0.287,Y -611.215,Z 974.310,A 0.000,B 0.000,C 90.000,E1 271.718} C_DIS
LIN {X -0.062,Y -604.701,Z 974.308,A 0.000,B 0.000,C 90.000,E1 271.375} C_DIS
LIN {X -0.085,Y -597.838,Z 974.306,A 0.000,B 0.000,C 90.000,E1 271.031} C_DIS
LIN {X 0.291,Y -590.556,Z 974.304,A 0.000,B 0.000,C 90.000,E1 270.688} C_DIS
LIN {X -0.039,Y -585.185,Z 974.303,A 0.000,B 0.000,C 90.000,E1 270.516} C_DIS
LIN {X -0.027,Y -575.724,Z 974.301,A 0.000,B 0.000,C 90.000,E1 270.229} C_DIS
LIN {X 0.129,Y -572.211,Z 974.301,A 0.000,B 0.000,C 90.000,E1 270.115} C_DIS
LIN {X -0.096,Y -565.829,Z 974.300,A 0.000,B 0.000,C 90.000,E1 270.000} C_DIS
LIN {X 0.101,Y -563.471,Z 974.300,A 0.000,B 0.000,C 90.000,E1 269.943} C_DIS
LIN {X 0.125,Y -557.783,Z 974.299,A 0.000,B 0.000,C 90.000,E1 269.885} C_DIS
LIN {X 0.084,Y -545.256,Z 974.299,A 0.000,B 0.000,C 90.000,E1 269.885} C_DIS
LIN {X -0.175,Y -543.574,Z 974.299,A 0.000,B 0.000,C 90.000,E1 269.885} C_DIS
LIN {X -0.219,Y -543.167,Z 974.299,A 0.000,B 0.000,C 90.000,E1 269.885} C_DIS
LIN {X 0.168,Y -542.752,Z 974.298,A 0.000,B 0.000,C 90.000,E1 269.656} C_DIS
LIN {X 0.091,Y -541.367,Z 974.288,A 0.000,B 0.000,C 90.000,E1 267.822} C_DIS
LIN {X -0.250,Y -540.004,Z 974.277,A 0.000,B 0.000,C 90.000,E1 265.869} C_DIS
LIN {X -0.164,Y -539.202,Z 974.271,A 0.000,B 0.000,C 90.000,E1 264.723} C_DIS
LIN {X 0.010,Y -538.103,Z 974.263,A 0.000,B 0.000,C 90.000,E1 263.280} C_DIS
LIN {X 0.164,Y -536.777,Z 974.255,A 0.000,B 0.000,C 90.000,E1 261.837} C_DIS
LIN {X -0.050,Y -534.752,Z 974.244,A 0.000,B 0.000,C 90.000,E1 259.859} C_DIS
LIN {X 0.109,Y -533.080,Z 974.236,A 0.000,B 0.000,C 90.000,E1 258.409} C_DIS
LIN {X -0.114,Y -531.814,Z 974.229,A 0.000,B 0.000,C 90.000,E1 257.285} C_DIS
LIN {X -0.234,Y -529.329,Z 974.218,A 0.000,B 0.000,C 90.000,E1 255.283} C_DIS
LIN {X 0.195,Y -527.516,Z 974.208,A 0.000,B 0.000,C 90.000,E1 253.504} C_DIS
LIN {X 0.217,Y -525.964,Z 974.201,A 0.000,B 0.000,C 90.000,E1 252.054} C_DIS
LIN {X 0.214,Y -524.121,Z 974.192,A 0.000,B 0.000,C 90.000,E1 250.604} C_DIS
LIN {X -0.164,Y -521.828,Z 974.183,A 0.000,B 0.000,C 90.000,E1 248.901} C_DIS
LIN {X 0.121,Y -520.001,Z 974.175,A 0.000,B 0.000,C 90.000,E1 247.411} C_DIS
LIN {X 0.087,Y -518.772,Z 974.170,A 0.000,B 0.000,C 90.000,E1 246.538} C_DIS
LIN {X -0.163,Y -516.590,Z 974.162,A 0.000,B 0.000,C 90.000,E1 245.101} C_DIS
LIN {X -0.237,Y -514.289,Z 974.153,A 0.000,B 0.000,C 90.000,E1 243.640} C_DIS
LIN {X -0.120,Y -512.958,Z 974.149,A 0.000,B 0.000,C 90.000,E1 242.743} C_DIS
LIN {X -0.145,Y -510.024,Z 974.139,A 0.000,B 0.000,C 90.000,E1 240.973} C_DIS
LIN {X 0.134,Y -507.416,Z 974.130,A 0.000,B 0.000,C 90.000,E1 239.459} C_DIS
LIN {X 0.034,Y -505.098,Z 974.124,A 0.000,B 0.000,C 90.000,E1 238.280} C_DIS
LIN {X -0.269,Y -502.687,Z 974.117,A 0.000,B 0.000,C 90.000,E1 237.120} C_DIS
LIN {X -0.204,Y -500.725,Z 974.112,A 0.000,B 0.000,C 90.000,E1 236.215} C_DIS
LIN {X -0.004,Y -497.271,Z 974.104,A 0.000,B 0.000,C 90.000,E1 234.689} C_DIS
LIN {X -0.277,Y -493.858,Z 974.095,A 0.000,B 0.000,C 90.000,E1 233.210} C_DIS
LIN {X -0.172,Y -489.651,Z 974.085,A 0.000,B 0.000,C 90.000,E1 231.376} C_DIS
LIN {X -0.162,Y -485.326,Z 974.075,A 0.000,B 0.000,C 90.000,E1 229.542} C_DIS
LIN {X -0.184,Y -480.407,Z 974.063,A 0.000,B 0.000,C 90.000,E1 227.391} C_DIS
LIN {X -0.018,Y -475.705,Z 974.051,A 0.000,B 0.000,C 90.000,E1 225.202} C_DIS
LIN {X -0.071,Y -471.581,Z 974.041,A 0.000,B 0.000,C 90.000,E1 223.338} C_DIS
LIN {X -0.131,Y -466.754,Z 974.029,A 0.000,B 0.000,C 90.000,E1 221.148} C_DIS
LIN {X -0.086,Y -463.217,Z 974.020,A 0.000,B 0.000,C 90.000,E1 219.564} C_DIS
LIN {X 0.087,Y -458.214,Z 974.007,A 0.000,B 0.000,C 90.000,E1 217.317} C_DIS
LIN {X 0.128,Y -453.988,Z 973.997,A 0.000,B 0.000,C 90.000,E1 215.391} C_DIS
LIN {X -0.197,Y -449.749,Z 973.986,A 0.000,B 0.000,C 90.000,E1 213.499} C_DIS
LIN {X -0.116,Y -445.515,Z 973.975,A 0.000,B 0.000,C 90.000,E1 211.544} C_DIS
LIN {X 0.193,Y -442.052,Z 973.966,A 0.000,B 0.000,C 90.000,E1 209.873} C_DIS
LIN {X 0.169,Y -439.140,Z 973.959,A 0.000,B 0.000,C 90.000,E1 208.565} C_DIS
LIN {X -0.055,Y -434.831,Z 973.948,A 0.000,B 0.000,C 90.000,E1 206.616} C_DIS
LIN {X -0.003,Y -431.870,Z 973.940,A 0.000,B 0.000,C 90.000,E1 205.283} C_DIS
LIN {X -0.191,Y -427.958,Z 973.931,A 0.000,B 0.000,C 90.000,E1 203.643} C_DIS
LIN {X 0.113,Y -423.464,Z 973.920,A 0.000,B 0.000,C 90.000,E1 201.589} C_DIS
LIN {X 0.168,Y -418.433,Z 973.907,A 0.000,B 0.000,C 90.000,E1 199.214} C_DIS
LIN {X 0.095,Y -413.014,Z 973.892,A 0.000,B 0.000,C 90.000,E1 196.496} C_DIS
LIN {X -0.236,Y -409.191,Z 973.880,A 0.000,B 0.000,C 90.000,E1 194.481} C_DIS
LIN {X 0.036,Y -405.906,Z 973.871,A 0.000,B 0.000,C 90.000,E1 192.715} C_DIS
LIN {X -0.163,Y -402.562,Z 973.861,A 0.000,B 0.000,C 90.000,E1 191.007} C_DIS
LIN {X -0.182,Y -399.952,Z 973.853,A 0.000,B 0.000,C 90.000,E1 189.613} C_DIS
LIN {X -0.165,Y -393.055,Z 973.832,A 0.000,B 0.000,C 90.000,E1 185.739} C_DIS
LIN {X -0.036,Y -391.457,Z 973.824,A 0.000,B 0.000,C 90.000,E1 184.302} C_DIS
LIN {X -0.093,Y -391.161,Z 973.822,A 0.000,B 0.000,C 90.000,E1 183.955} C_DIS
LIN {X 0.128,Y -390.910,Z 973.818,A 0.000,B 0.000,C 90.000,E1 183.212} C_DIS
LIN {X -0.020,Y -391.242,Z 973.814,A 0.000,B 0.000,C 90.000,E1 182.522} C_DIS
LIN {X -0.145,Y -392.065,Z 973.811,A 0.000,B 0.000,C 90.000,E1 182.007} C_DIS
LIN {X 0.140,Y -393.449,Z 973.808,A 0.000,B 0.000,C 90.000,E1 181.432} C_DIS
LIN {X 0.028,Y -395.497,Z 973.805,A 0.000,B 0.000,C 90.000,E1 180.917} C_DIS
LIN {X 0.047,Y -398.037,Z 973.803,A 0.000,B 0.000,C 90.000,E1 180.458} C_DIS
LIN {X -0.014,Y -400.314,Z 973.801,A 0.000,B 0.000,C 90.000,E1 180.115} C_DIS
LIN {X -0.107,Y -405.040,Z 973.797,A 0.000,B 0.000,C 90.000,E1 179.542} C_DIS
LIN {X -0.006,Y -410.993,Z 973.794,A 0.000,B 0.000,C 90.000,E1 178.912} C_DIS
LIN {X 0.073,Y -419.939,Z 973.789,A 0.000,B 0.000,C 90.000,E1 178.051} C_DIS
LIN {X 0.016,Y -427.435,Z 973.785,A 0.000,B 0.000,C 90.000,E1 177.364} C_DIS
LIN {X 0.078,Y -437.616,Z 973.780,A 0.000,B 0.000,C 90.000,E1 176.388} C_DIS
LIN {X -0.220,Y -447.883,Z 973.774,A 0.000,B 0.000,C 90.000,E1 175.412} C_DIS
LIN {X 0.128,Y -459.342,Z 973.768,A 0.000,B 0.000,C 90.000,E1 174.204} C_DIS
LIN {X -0.245,Y -466.114,Z 973.764,A 0.000,B 0.000,C 90.000,E1 173.514} C_DIS
LIN {X 0.068,Y -471.519,Z 973.760,A 0.000,B 0.000,C 90.000,E1 172.875} C_DIS
LIN {X 0.122,Y -480.480,Z 973.754,A 0.000,B 0.000,C 90.000,E1 171.781} C_DIS
LIN {X -0.037,Y -486.697,Z 973.750,A 0.000,B 0.000,C 90.000,E1 171.027} C_DIS
LIN {X -0.187,Y -494.864,Z 973.744,A 0.000,B 0.000,C 90.000,E1 169.982} C_DIS
LIN {X -0.182,Y -502.529,Z 973.738,A 0.000,B 0.000,C 90.000,E1 168.926} C_DIS
LIN {X -0.150,Y -509.725,Z 973.733,A 0.000,B 0.000,C 90.000,E1 167.881} C_DIS
LIN {X 0.056,Y -518.521,Z 973.725,A 0.000,B 0.000,C 90.000,E1 166.533} C_DIS
LIN {X -0.151,Y -521.374,Z 973.723,A 0.000,B 0.000,C 90.000,E1 166.117} C_DIS
LIN {X -0.195,Y -527.513,Z 973.717,A 0.000,B 0.000,C 90.000,E1 165.102} C_DIS
LIN {X 0.017,Y -532.959,Z 973.712,A 0.000,B 0.000,C 90.000,E1 164.212} C_DIS
LIN {X 0.135,Y -538.966,Z 973.707,A 0.000,B 0.000,C 90.000,E1 163.196} C_DIS
LIN {X -0.191,Y -544.789,Z 973.701,A 0.000,B 0.000,C 90.000,E1 162.236} C_DIS
LIN {X 0.208,Y -552.986,Z 973.693,A 0.000,B 0.000,C 90.000,E1 160.786} C_DIS
LIN {X -0.071,Y -559.343,Z 973.687,A 0.000,B 0.000,C 90.000,E1 159.699} C_DIS
LIN {X -0.289,Y -563.134,Z 973.683,A 0.000,B 0.000,C 90.000,E1 159.028} C_DIS
LIN {X 0.065,Y -568.238,Z 973.678,A 0.000,B 0.000,C 90.000,E1 158.028} C_DIS
LIN {X -0.166,Y -572.422,Z 973.673,A 0.000,B 0.000,C 90.000,E1 157.230} C_DIS
LIN {X -0.133,Y -576.461,Z 973.669,A 0.000,B 0.000,C 90.000,E1 156.410} C_DIS
LIN {X -0.291,Y -580.304,Z 973.664,A 0.000,B 0.000,C 90.000,E1 155.613} C_DIS
LIN {X -0.179,Y -583.914,Z 973.660,A 0.000,B 0.000,C 90.000,E1 154.793} C_DIS
LIN {X -0.151,Y -588.304,Z 973.654,A 0.000,B 0.000,C 90.000,E1 153.717} C_DIS
LIN {X 0.305,Y -591.363,Z 973.649,A 0.000,B 0.000,C 90.000,E1 152.871} C_DIS
LIN {X -0.097,Y -595.038,Z 973.644,A 0.000,B 0.000,C 90.000,E1 151.847} C_DIS
LIN {X 0.038,Y -599.204,Z 973.636,A 0.000,B 0.000,C 90.000,E1 150.511} C_DIS
LIN {X -0.119,Y -604.143,Z 973.628,A 0.000,B 0.000,C 90.000,E1 148.948} C_DIS
LIN {X -0.073,Y -609.068,Z 973.619,A 0.000,B 0.000,C 90.000,E1 147.375} C_DIS
LIN {X 0.082,Y -613.867,Z 973.610,A 0.000,B 0.000,C 90.000,E1 145.801} C_DIS
LIN {X -0.131,Y -617.917,Z 973.603,A 0.000,B 0.000,C 90.000,E1 144.529} C_DIS
LIN {X 0.225,Y -621.896,Z 973.596,A 0.000,B 0.000,C 90.000,E1 143.210} C_DIS
LIN {X -0.170,Y -627.374,Z 973.586,A 0.000,B 0.000,C 90.000,E1 141.457} C_DIS
LIN {X 0.213,Y -631.275,Z 973.579,A 0.000,B 0.000,C 90.000,E1 140.150} C_DIS
LIN {X -0.313,Y -635.048,Z 973.572,A 0.000,B 0.000,C 90.000,E1 138.933} C_DIS
LIN {X -0.150,Y -641.260,Z 973.561,A 0.000,B 0.000,C 90.000,E1 136.905} C_DIS
LIN {X -0.149,Y -646.055,Z 973.552,A 0.000,B 0.000,C 90.000,E1 135.405} C_DIS
LIN {X -0.246,Y -654.429,Z 973.538,A 0.000,B 0.000,C 90.000,E1 132.933} C_DIS
LIN {X -0.009,Y -662.460,Z 973.526,A 0.000,B 0.000,C 90.000,E1 130.701} C_DIS
LIN {X -0.029,Y -667.008,Z 973.519,A 0.000,B 0.000,C 90.000,E1 129.483} C_DIS
LIN {X 0.111,Y -672.134,Z 973.511,A 0.000,B 0.000,C 90.000,E1 128.016} C_DIS
LIN {X 0.344,Y -676.112,Z 973.505,A 0.000,B 0.000,C 90.000,E1 126.790} C_DIS
LIN {X 0.241,Y -679.834,Z 973.498,A 0.000,B 0.000,C 90.000,E1 125.598} C_DIS
LIN {X 0.201,Y -683.446,Z 973.491,A 0.000,B 0.000,C 90.000,E1 124.405} C_DIS
LIN {X -0.167,Y -686.797,Z 973.485,A 0.000,B 0.000,C 90.000,E1 123.245} C_DIS
LIN {X -0.116,Y -689.859,Z 973.478,A 0.000,B 0.000,C 90.000,E1 122.054} C_DIS
LIN {X -0.397,Y -692.270,Z 973.473,A 0.000,B 0.000,C 90.000,E1 121.131} C_DIS
LIN {X 0.307,Y -694.407,Z 973.468,A 0.000,B 0.000,C 90.000,E1 120.129} C_DIS
LIN {X -0.161,Y -695.804,Z 973.464,A 0.000,B 0.000,C 90.000,E1 119.461} C_DIS
LIN {X -0.011,Y -696.877,Z 973.460,A 0.000,B 0.000,C 90.000,E1 118.743} C_DIS
LIN {X 0.149,Y -697.729,Z 973.456,A 0.000,B 0.000,C 90.000,E1 118.025} C_DIS
LIN {X 0.173,Y -699.122,Z 973.448,A 0.000,B 0.000,C 90.000,E1 116.616} C_DIS
LIN {X -0.048,Y -699.949,Z 973.441,A 0.000,B 0.000,C 90.000,E1 115.463} C_DIS
LIN {X -0.170,Y -700.222,Z 973.438,A 0.000,B 0.000,C 90.000,E1 114.771} C_DIS
LIN {X 0.082,Y -700.282,Z 973.435,A 0.000,B 0.000,C 90.000,E1 114.283} C_DIS
LIN {X -0.018,Y -699.913,Z 973.432,A 0.000,B 0.000,C 90.000,E1 113.823} C_DIS
LIN {X -0.031,Y -699.607,Z 973.431,A 0.000,B 0.000,C 90.000,E1 113.590} C_DIS
LIN {X -0.143,Y -698.157,Z 973.428,A 0.000,B 0.000,C 90.000,E1 113.131} C_DIS
LIN {X -0.155,Y -697.093,Z 973.427,A 0.000,B 0.000,C 90.000,E1 112.898} C_DIS
LIN {X 0.227,Y -694.104,Z 973.425,A 0.000,B 0.000,C 90.000,E1 112.514} C_DIS
LIN {X 0.208,Y -691.808,Z 973.424,A 0.000,B 0.000,C 90.000,E1 112.280} C_DIS
LIN {X -0.311,Y -689.999,Z 973.423,A 0.000,B 0.000,C 90.000,E1 112.206} C_DIS
LIN {X 0.229,Y -685.383,Z 973.422,A 0.000,B 0.000,C 90.000,E1 111.972} C_DIS
LIN {X 0.136,Y -680.653,Z 973.421,A 0.000,B 0.000,C 90.000,E1 111.844} C_DIS
LIN {X 0.277,Y -675.532,Z 973.421,A 0.000,B 0.000,C 90.000,E1 111.716} C_DIS
LIN {X 0.015,Y -670.369,Z 973.421,A 0.000,B 0.000,C 90.000,E1 111.716} C_DIS
LIN {X -0.019,Y -626.340,Z 973.421,A 0.000,B 0.000,C 90.000,E1 111.716} C_DIS
LIN {X -0.142,Y -621.353,Z 973.420,A 0.000,B 0.000,C 90.000,E1 111.642} C_DIS
LIN {X 0.140,Y -615.570,Z 973.419,A 0.000,B 0.000,C 90.000,E1 111.482} C_DIS
LIN {X -0.094,Y -610.159,Z 973.419,A 0.000,B 0.000,C 90.000,E1 111.334} C_DIS
LIN {X 0.069,Y -603.612,Z 973.417,A 0.000,B 0.000,C 90.000,E1 111.046} C_DIS
LIN {X -0.103,Y -597.542,Z 973.415,A 0.000,B 0.000,C 90.000,E1 110.737} C_DIS
LIN {X -0.057,Y -591.677,Z 973.413,A 0.000,B 0.000,C 90.000,E1 110.355} C_DIS
LIN {X -0.273,Y -583.485,Z 973.410,A 0.000,B 0.000,C 90.000,E1 109.758} C_DIS
LIN {X -0.173,Y -576.354,Z 973.407,A 0.000,B 0.000,C 90.000,E1 109.195} C_DIS
LIN {X -0.204,Y -574.898,Z 973.406,A 0.000,B 0.000,C 90.000,E1 109.087} C_DIS
LIN {X 0.279,Y -566.673,Z 973.403,A 0.000,B 0.000,C 90.000,E1 108.544} C_DIS
LIN {X 0.125,Y -553.165,Z 973.399,A 0.000,B 0.000,C 90.000,E1 107.873} C_DIS
LIN {X -0.171,Y -551.832,Z 973.399,A 0.000,B 0.000,C 90.000,E1 107.819} C_DIS
LIN {X 0.046,Y -550.043,Z 973.398,A 0.000,B 0.000,C 90.000,E1 107.638} C_DIS
LIN {X 0.010,Y -550.031,Z 973.398,A 0.000,B 0.000,C 90.000,E1 107.638} C_DIS
LIN {X 0.120,Y -549.646,Z 973.397,A 0.000,B 0.000,C 90.000,E1 107.457} C_DIS
LIN {X -0.053,Y -549.555,Z 973.394,A 0.000,B 0.000,C 90.000,E1 106.913} C_DIS
LIN {X 0.218,Y -550.156,Z 973.386,A 0.000,B 0.000,C 90.000,E1 105.481} C_DIS
LIN {X -0.264,Y -551.444,Z 973.372,A 0.000,B 0.000,C 90.000,E1 103.008} C_DIS
LIN {X -0.025,Y -554.073,Z 973.355,A 0.000,B 0.000,C 90.000,E1 99.905} C_DIS
LIN {X 0.092,Y -555.767,Z 973.346,A 0.000,B 0.000,C 90.000,E1 98.219} C_DIS
LIN {X 0.029,Y -557.050,Z 973.338,A 0.000,B 0.000,C 90.000,E1 96.834} C_DIS
LIN {X -0.140,Y -557.968,Z 973.332,A 0.000,B 0.000,C 90.000,E1 95.739} C_DIS
LIN {X 0.258,Y -558.765,Z 973.326,A 0.000,B 0.000,C 90.000,E1 94.588} C_DIS
LIN {X 0.270,Y -559.802,Z 973.316,A 0.000,B 0.000,C 90.000,E1 92.922} C_DIS
LIN {X 0.182,Y -560.528,Z 973.309,A 0.000,B 0.000,C 90.000,E1 91.547} C_DIS
LIN {X 0.193,Y -561.311,Z 973.299,A 0.000,B 0.000,C 90.000,E1 89.885} C_DIS
LIN {X 0.120,Y -561.728,Z 973.292,A 0.000,B 0.000,C 90.000,E1 88.511} C_DIS
LIN {X 0.160,Y -562.106,Z 973.283,A 0.000,B 0.000,C 90.000,E1 86.849} C_DIS
LIN {X 0.145,Y -562.325,Z 973.275,A 0.000,B 0.000,C 90.000,E1 85.469} C_DIS
LIN {X -0.193,Y -562.581,Z 973.264,A 0.000,B 0.000,C 90.000,E1 83.571} C_DIS
LIN {X 0.240,Y -562.997,Z 973.252,A 0.000,B 0.000,C 90.000,E1 81.319} C_DIS
LIN {X -0.245,Y -563.805,Z 973.240,A 0.000,B 0.000,C 90.000,E1 79.162} C_DIS
LIN {X -0.031,Y -564.890,Z 973.227,A 0.000,B 0.000,C 90.000,E1 76.937} C_DIS
LIN {X 0.168,Y -566.184,Z 973.217,A 0.000,B 0.000,C 90.000,E1 74.991} C_DIS
LIN {X -0.009,Y -567.504,Z 973.206,A 0.000,B 0.000,C 90.000,E1 73.087} C_DIS
LIN {X 0.049,Y -568.402,Z 973.198,A 0.000,B 0.000,C 90.000,E1 71.710} C_DIS
LIN {X -0.082,Y -569.518,Z 973.188,A 0.000,B 0.000,C 90.000,E1 69.806} C_DIS
LIN {X 0.192,Y -570.183,Z 973.180,A 0.000,B 0.000,C 90.000,E1 68.411} C_DIS
LIN {X 0.146,Y -570.721,Z 973.173,A 0.000,B 0.000,C 90.000,E1 67.050} C_DIS
LIN {X -0.016,Y -571.114,Z 973.167,A 0.000,B 0.000,C 90.000,E1 65.973} C_DIS
LIN {X 0.186,Y -571.538,Z 973.159,A 0.000,B 0.000,C 90.000,E1 64.588} C_DIS
LIN {X -0.125,Y -571.875,Z 973.151,A 0.000,B 0.000,C 90.000,E1 63.256} C_DIS
LIN {X -0.176,Y -572.130,Z 973.144,A 0.000,B 0.000,C 90.000,E1 61.897} C_DIS
LIN {X -0.112,Y -572.285,Z 973.135,A 0.000,B 0.000,C 90.000,E1 60.255} C_DIS
LIN {X -0.053,Y -572.452,Z 973.126,A 0.000,B 0.000,C 90.000,E1 58.614} C_DIS
LIN {X 0.118,Y -572.624,Z 973.117,A 0.000,B 0.000,C 90.000,E1 56.962} C_DIS
LIN {X 0.165,Y -572.550,Z 973.109,A 0.000,B 0.000,C 90.000,E1 55.595} C_DIS
LIN {X 0.252,Y -572.467,Z 973.104,A 0.000,B 0.000,C 90.000,E1 54.769} C_DIS
LIN {X 0.007,Y -572.111,Z 973.098,A 0.000,B 0.000,C 90.000,E1 53.703} C_DIS
LIN {X -0.242,Y -571.622,Z 973.092,A 0.000,B 0.000,C 90.000,E1 52.637} C_DIS
LIN {X -0.286,Y -571.151,Z 973.088,A 0.000,B 0.000,C 90.000,E1 51.823} C_DIS
LIN {X -0.198,Y -570.355,Z 973.082,A 0.000,B 0.000,C 90.000,E1 50.723} C_DIS
LIN {X -0.128,Y -569.259,Z 973.076,A 0.000,B 0.000,C 90.000,E1 49.622} C_DIS
LIN {X -0.134,Y -567.991,Z 973.070,A 0.000,B 0.000,C 90.000,E1 48.528} C_DIS
LIN {X -0.219,Y -566.837,Z 973.065,A 0.000,B 0.000,C 90.000,E1 47.715} C_DIS
LIN {X -0.257,Y -565.039,Z 973.059,A 0.000,B 0.000,C 90.000,E1 46.620} C_DIS
LIN {X 0.069,Y -562.813,Z 973.053,A 0.000,B 0.000,C 90.000,E1 45.486} C_DIS
LIN {X 0.222,Y -561.615,Z 973.050,A 0.000,B 0.000,C 90.000,E1 44.919} C_DIS
LIN {X 0.038,Y -559.502,Z 973.045,A 0.000,B 0.000,C 90.000,E1 44.109} C_DIS
LIN {X 0.164,Y -557.998,Z 973.042,A 0.000,B 0.000,C 90.000,E1 43.542} C_DIS
LIN {X 0.344,Y -555.439,Z 973.037,A 0.000,B 0.000,C 90.000,E1 42.690} C_DIS
LIN {X 0.063,Y -553.631,Z 973.034,A 0.000,B 0.000,C 90.000,E1 42.162} C_DIS
LIN {X 0.199,Y -550.485,Z 973.030,A 0.000,B 0.000,C 90.000,E1 41.310} C_DIS
LIN {X 0.294,Y -547.013,Z 973.025,A 0.000,B 0.000,C 90.000,E1 40.458} C_DIS
LIN {X -0.196,Y -543.918,Z 973.021,A 0.000,B 0.000,C 90.000,E1 39.806} C_DIS
LIN {X 0.235,Y -539.788,Z 973.016,A 0.000,B 0.000,C 90.000,E1 38.910} C_DIS
LIN {X -0.136,Y -533.695,Z 973.010,A 0.000,B 0.000,C 90.000,E1 37.810} C_DIS
LIN {X -0.170,Y -527.108,Z 973.004,A 0.000,B 0.000,C 90.000,E1 36.664} C_DIS
LIN {X 0.123,Y -520.126,Z 972.997,A 0.000,B 0.000,C 90.000,E1 35.471} C_DIS
LIN {X -0.116,Y -512.489,Z 972.991,A 0.000,B 0.000,C 90.000,E1 34.326} C_DIS
LIN {X 0.141,Y -508.262,Z 972.987,A 0.000,B 0.000,C 90.000,E1 33.706} C_DIS
LIN {X 0.056,Y -500.256,Z 972.982,A 0.000,B 0.000,C 90.000,E1 32.673} C_DIS
LIN {X 0.025,Y -493.780,Z 972.977,A 0.000,B 0.000,C 90.000,E1 31.926} C_DIS
LIN {X -0.175,Y -487.117,Z 972.973,A 0.000,B 0.000,C 90.000,E1 31.209} C_DIS
LIN {X 0.251,Y -481.430,Z 972.970,A 0.000,B 0.000,C 90.000,E1 30.590} C_DIS
LIN {X -0.003,Y -474.325,Z 972.966,A 0.000,B 0.000,C 90.000,E1 29.922} C_DIS
LIN {X 0.056,Y -468.454,Z 972.963,A 0.000,B 0.000,C 90.000,E1 29.361} C_DIS
LIN {X -0.072,Y -459.610,Z 972.959,A 0.000,B 0.000,C 90.000,E1 28.565} C_DIS
LIN {X -0.060,Y -450.488,Z 972.954,A 0.000,B 0.000,C 90.000,E1 27.769} C_DIS
LIN {X 0.106,Y -430.736,Z 972.945,A 0.000,B 0.000,C 90.000,E1 26.052} C_DIS
LIN {X -0.103,Y -415.893,Z 972.937,A 0.000,B 0.000,C 90.000,E1 24.719} C_DIS
LIN {X -0.093,Y -404.438,Z 972.931,A 0.000,B 0.000,C 90.000,E1 23.567} C_DIS
LIN {X 0.079,Y -397.499,Z 972.927,A 0.000,B 0.000,C 90.000,E1 22.770} C_DIS
LIN {X 0.036,Y -393.516,Z 972.923,A 0.000,B 0.000,C 90.000,E1 22.206} C_DIS
LIN {X -0.094,Y -391.141,Z 972.921,A 0.000,B 0.000,C 90.000,E1 21.716} C_DIS
LIN {X -0.039,Y -390.015,Z 972.918,A 0.000,B 0.000,C 90.000,E1 21.153} C_DIS
LIN {X 0.060,Y -389.873,Z 972.913,A 0.000,B 0.000,C 90.000,E1 20.248} C_DIS
LIN {X -0.184,Y -390.513,Z 972.907,A 0.000,B 0.000,C 90.000,E1 19.214} C_DIS
LIN {X 0.190,Y -393.250,Z 972.891,A 0.000,B 0.000,C 90.000,E1 16.315} C_DIS
LIN {X -0.102,Y -397.201,Z 972.873,A 0.000,B 0.000,C 90.000,E1 13.175} C_DIS
LIN {X -0.145,Y -403.002,Z 972.852,A 0.000,B 0.000,C 90.000,E1 9.321} C_DIS
LIN {X -0.200,Y -406.100,Z 972.842,A 0.000,B 0.000,C 90.000,E1 7.587} C_DIS
LIN {X -0.179,Y -411.477,Z 972.827,A 0.000,B 0.000,C 90.000,E1 4.816} C_DIS
LIN {X -0.141,Y -415.882,Z 972.815,A 0.000,B 0.000,C 90.000,E1 2.751} C_DIS
LIN {X -0.007,Y -420.658,Z 972.804,A 0.000,B 0.000,C 90.000,E1 0.688} C_DIS
LIN {X 0.000,Y -422.789,Z 972.800,A 0.000,B 0.000,C 90.000,E1 360.000} C_DIS
LIN {X 0.183,Y -424.505,Z 972.798,A 0.000,B 0.000,C 90.000,E1 359.599} C_DIS
LIN {X -0.127,Y -426.465,Z 972.796,A 0.000,B 0.000,C 90.000,E1 359.312} C_DIS
LIN {X 0.181,Y -429.670,Z 972.794,A 0.000,B 0.000,C 90.000,E1 358.854} C_DIS
LIN {X -0.180,Y -433.677,Z 972.792,A 0.000,B 0.000,C 90.000,E1 358.568} C_DIS
LIN {X 0.149,Y -435.573,Z 972.791,A 0.000,B 0.000,C 90.000,E1 358.396} C_DIS
LIN {X 0.205,Y -447.904,Z 972.787,A 0.000,B 0.000,C 90.000,E1 357.707} C_DIS
LIN {X -0.086,Y -461.197,Z 972.783,A 0.000,B 0.000,C 90.000,E1 357.020} C_DIS
LIN {X 0.072,Y -477.804,Z 972.778,A 0.000,B 0.000,C 90.000,E1 356.102} C_DIS
LIN {X 0.223,Y -490.569,Z 972.774,A 0.000,B 0.000,C 90.000,E1 355.355} C_DIS
LIN {X -0.101,Y -502.084,Z 972.771,A 0.000,B 0.000,C 90.000,E1 354.723} C_DIS
LIN {X -0.131,Y -509.850,Z 972.768,A 0.000,B 0.000,C 90.000,E1 354.261} C_DIS
LIN {X 0.045,Y -519.182,Z 972.765,A 0.000,B 0.000,C 90.000,E1 353.628} C_DIS
LIN {X -0.113,Y -526.943,Z 972.762,A 0.000,B 0.000,C 90.000,E1 353.109} C_DIS
LIN {X 0.023,Y -534.292,Z 972.759,A 0.000,B 0.000,C 90.000,E1 352.534} C_DIS
LIN {X -0.110,Y -541.418,Z 972.755,A 0.000,B 0.000,C 90.000,E1 351.951} C_DIS
LIN {X -0.140,Y -548.220,Z 972.752,A 0.000,B 0.000,C 90.000,E1 351.319} C_DIS
LIN {X 0.229,Y -554.611,Z 972.748,A 0.000,B 0.000,C 90.000,E1 350.622} C_DIS
LIN {X 0.254,Y -560.173,Z 972.745,A 0.000,B 0.000,C 90.000,E1 349.982} C_DIS
LIN {X -0.252,Y -565.600,Z 972.741,A 0.000,B 0.000,C 90.000,E1 349.342} C_DIS
LIN {X -0.047,Y -570.612,Z 972.737,A 0.000,B 0.000,C 90.000,E1 348.634} C_DIS
LIN {X -0.101,Y -573.412,Z 972.735,A 0.000,B 0.000,C 90.000,E1 348.229} C_DIS
LIN {X 0.183,Y -577.745,Z 972.731,A 0.000,B 0.000,C 90.000,E1 347.521} C_DIS
LIN {X 0.044,Y -583.290,Z 972.726,A 0.000,B 0.000,C 90.000,E1 346.589} C_DIS
LIN {X 0.333,Y -587.670,Z 972.721,A 0.000,B 0.000,C 90.000,E1 345.755} C_DIS
LIN {X -0.046,Y -591.841,Z 972.717,A 0.000,B 0.000,C 90.000,E1 344.991} C_DIS
LIN {X 0.110,Y -596.442,Z 972.711,A 0.000,B 0.000,C 90.000,E1 344.047} C_DIS
LIN {X -0.088,Y -600.864,Z 972.706,A 0.000,B 0.000,C 90.000,E1 343.142} C_DIS
LIN {X -0.229,Y -605.030,Z 972.701,A 0.000,B 0.000,C 90.000,E1 342.236} C_DIS
LIN {X 0.217,Y -609.419,Z 972.695,A 0.000,B 0.000,C 90.000,E1 341.148} C_DIS
LIN {X 0.149,Y -613.638,Z 972.690,A 0.000,B 0.000,C 90.000,E1 340.115} C_DIS
LIN {X 0.135,Y -617.531,Z 972.684,A 0.000,B 0.000,C 90.000,E1 339.082} C_DIS
LIN {X 0.148,Y -621.977,Z 972.677,A 0.000,B 0.000,C 90.000,E1 337.794} C_DIS
LIN {X -0.110,Y -625.305,Z 972.671,A 0.000,B 0.000,C 90.000,E1 336.794} C_DIS
LIN {X -0.322,Y -628.478,Z 972.665,A 0.000,B 0.000,C 90.000,E1 335.793} C_DIS
LIN {X 0.102,Y -632.091,Z 972.658,A 0.000,B 0.000,C 90.000,E1 334.485} C_DIS
LIN {X 0.167,Y -633.453,Z 972.656,A 0.000,B 0.000,C 90.000,E1 333.973} C_DIS
LIN {X -0.148,Y -637.141,Z 972.647,A 0.000,B 0.000,C 90.000,E1 332.487} C_DIS
LIN {X -0.082,Y -640.439,Z 972.639,A 0.000,B 0.000,C 90.000,E1 330.973} C_DIS
LIN {X 0.161,Y -642.496,Z 972.633,A 0.000,B 0.000,C 90.000,E1 329.950} C_DIS
LIN {X -0.298,Y -644.824,Z 972.626,A 0.000,B 0.000,C 90.000,E1 328.742} C_DIS
LIN {X 0.104,Y -646.362,Z 972.621,A 0.000,B 0.000,C 90.000,E1 327.709} C_DIS
LIN {X 0.182,Y -647.821,Z 972.615,A 0.000,B 0.000,C 90.000,E1 326.707} C_DIS
LIN {X 0.092,Y -649.034,Z 972.610,A 0.000,B 0.000,C 90.000,E1 325.722} C_DIS
LIN {X -0.347,Y -650.048,Z 972.604,A 0.000,B 0.000,C 90.000,E1 324.769} C_DIS
LIN {X 0.033,Y -651.140,Z 972.597,A 0.000,B 0.000,C 90.000,E1 323.497} C_DIS
LIN {X 0.379,Y -651.865,Z 972.592,A 0.000,B 0.000,C 90.000,E1 322.477} C_DIS
LIN {X -0.178,Y -652.457,Z 972.586,A 0.000,B 0.000,C 90.000,E1 321.537} C_DIS
LIN {X 0.185,Y -652.946,Z 972.581,A 0.000,B 0.000,C 90.000,E1 320.517} C_DIS
LIN {X 0.396,Y -653.749,Z 972.571,A 0.000,B 0.000,C 90.000,E1 318.771} C_DIS
LIN {X -0.005,Y -655.648,Z 972.556,A 0.000,B 0.000,C 90.000,E1 316.095} C_DIS
LIN {X 0.330,Y -656.381,Z 972.551,A 0.000,B 0.000,C 90.000,E1 315.081} C_DIS
LIN {X 0.079,Y -658.012,Z 972.540,A 0.000,B 0.000,C 90.000,E1 313.137} C_DIS
LIN {X -0.085,Y -659.445,Z 972.530,A 0.000,B 0.000,C 90.000,E1 311.434} C_DIS
LIN {X 0.335,Y -660.295,Z 972.523,A 0.000,B 0.000,C 90.000,E1 310.172} C_DIS
LIN {X -0.152,Y -661.087,Z 972.517,A 0.000,B 0.000,C 90.000,E1 308.991} C_DIS
LIN {X -0.144,Y -661.860,Z 972.508,A 0.000,B 0.000,C 90.000,E1 307.523} C_DIS
LIN {X -0.139,Y -662.175,Z 972.504,A 0.000,B 0.000,C 90.000,E1 306.790} C_DIS
LIN {X 0.012,Y -662.518,Z 972.496,A 0.000,B 0.000,C 90.000,E1 305.311} C_DIS
LIN {X -0.149,Y -663.019,Z 972.485,A 0.000,B 0.000,C 90.000,E1 303.372} C_DIS
LIN {X -0.027,Y -665.389,Z 972.464,A 0.000,B 0.000,C 90.000,E1 299.461} C_DIS
LIN {X 0.231,Y -670.490,Z 972.443,A 0.000,B 0.000,C 90.000,E1 295.796} C_DIS
LIN {X -0.086,Y -673.448,Z 972.434,A 0.000,B 0.000,C 90.000,E1 294.131} C_DIS
LIN {X 0.073,Y -675.030,Z 972.429,A 0.000,B 0.000,C 90.000,E1 293.153} C_DIS
LIN {X 0.251,Y -675.410,Z 972.427,A 0.000,B 0.000,C 90.000,E1 292.898} C_DIS
LIN {X -0.101,Y -675.863,Z 972.423,A 0.000,B 0.000,C 90.000,E1 292.206} C_DIS
LIN {X -0.002,Y -675.484,Z 972.421,A 0.000,B 0.000,C 90.000,E1 291.716} C_DIS
LIN {X 0.171,Y -675.049,Z 972.419,A 0.000,B 0.000,C 90.000,E1 291.461} C_DIS
LIN {X 0.266,Y -673.408,Z 972.417,A 0.000,B 0.000,C 90.000,E1 290.972} C_DIS
LIN {X 0.109,Y -672.876,Z 972.416,A 0.000,B 0.000,C 90.000,E1 290.865} C_DIS
LIN {X 0.192,Y -672.072,Z 972.415,A 0.000,B 0.000,C 90.000,E1 290.737} C_DIS
LIN {X 0.271,Y -670.872,Z 972.415,A 0.000,B 0.000,C 90.000,E1 290.610} C_DIS
LIN {X 0.116,Y -665.494,Z 972.412,A 0.000,B 0.000,C 90.000,E1 290.174} C_DIS
LIN {X 0.177,Y -654.165,Z 972.408,A 0.000,B 0.000,C 90.000,E1 289.450} C_DIS
LIN {X -0.036,Y -652.905,Z 972.407,A 0.000,B 0.000,C 90.000,E1 289.322} C_DIS
LIN {X -0.079,Y -652.886,Z 972.407,A 0.000,B 0.000,C 90.000,E1 289.322} C_DIS
LIN {X -0.165,Y -652.804,Z 972.407,A 0.000,B 0.000,C 90.000,E1 289.214} C_DIS
LIN {X -0.213,Y -654.502,Z 972.404,A 0.000,B 0.000,C 90.000,E1 288.725} C_DIS
LIN {X -0.294,Y -662.114,Z 972.397,A 0.000,B 0.000,C 90.000,E1 287.457} C_DIS
LIN {X 0.251,Y -666.094,Z 972.393,A 0.000,B 0.000,C 90.000,E1 286.677} C_DIS
LIN {X 0.084,Y -668.351,Z 972.390,A 0.000,B 0.000,C 90.000,E1 286.205} C_DIS
LIN {X 0.114,Y -670.208,Z 972.387,A 0.000,B 0.000,C 90.000,E1 285.717} C_DIS
LIN {X 0.042,Y -671.060,Z 972.386,A 0.000,B 0.000,C 90.000,E1 285.481} C_DIS
LIN {X -0.156,Y -673.059,Z 972.382,A 0.000,B 0.000,C 90.000,E1 284.773} C_DIS
LIN {X -0.333,Y -674.498,Z 972.378,A 0.000,B 0.000,C 90.000,E1 284.064} C_DIS
LIN {X 0.213,Y -675.270,Z 972.375,A 0.000,B 0.000,C 90.000,E1 283.536} C_DIS
LIN {X 0.109,Y -675.867,Z 972.373,A 0.000,B 0.000,C 90.000,E1 283.063} C_DIS
LIN {X -0.043,Y -676.441,Z 972.369,A 0.000,B 0.000,C 90.000,E1 282.355} C_DIS
LIN {X -0.143,Y -676.682,Z 972.366,A 0.000,B 0.000,C 90.000,E1 281.883} C_DIS
LIN {X 0.283,Y -676.699,Z 972.363,A 0.000,B 0.000,C 90.000,E1 281.366} C_DIS
LIN {X 0.182,Y -676.486,Z 972.361,A 0.000,B 0.000,C 90.000,E1 280.894} C_DIS
LIN {X -0.099,Y -675.738,Z 972.357,A 0.000,B 0.000,C 90.000,E1 280.197} C_DIS
LIN {X -0.213,Y -674.965,Z 972.354,A 0.000,B 0.000,C 90.000,E1 279.726} C_DIS
LIN {X 0.219,Y -673.856,Z 972.351,A 0.000,B 0.000,C 90.000,E1 279.208} C_DIS
LIN {X -0.017,Y -672.454,Z 972.349,A 0.000,B 0.000,C 90.000,E1 278.746} C_DIS
LIN {X -0.334,Y -669.880,Z 972.345,A 0.000,B 0.000,C 90.000,E1 278.049} C_DIS
LIN {X 0.074,Y -667.812,Z 972.342,A 0.000,B 0.000,C 90.000,E1 277.530} C_DIS
LIN {X -0.205,Y -664.627,Z 972.339,A 0.000,B 0.000,C 90.000,E1 276.947} C_DIS
LIN {X 0.160,Y -661.704,Z 972.336,A 0.000,B 0.000,C 90.000,E1 276.429} C_DIS
LIN {X -0.249,Y -657.392,Z 972.332,A 0.000,B 0.000,C 90.000,E1 275.853} C_DIS
LIN {X -0.039,Y -652.450,Z 972.329,A 0.000,B 0.000,C 90.000,E1 275.220} C_DIS
LIN {X 0.238,Y -648.171,Z 972.326,A 0.000,B 0.000,C 90.000,E1 274.702} C_DIS
LIN {X -0.209,Y -643.498,Z 972.324,A 0.000,B 0.000,C 90.000,E1 274.245} C_DIS
LIN {X 0.145,Y -638.571,Z 972.321,A 0.000,B 0.000,C 90.000,E1 273.726} C_DIS
LIN {X -0.056,Y -631.993,Z 972.318,A 0.000,B 0.000,C 90.000,E1 273.154} C_DIS
LIN {X 0.098,Y -624.966,Z 972.314,A 0.000,B 0.000,C 90.000,E1 272.579} C_DIS
LIN {X -0.058,Y -617.619,Z 972.311,A 0.000,B 0.000,C 90.000,E1 272.064} C_DIS
LIN {X -0.034,Y -611.363,Z 972.309,A 0.000,B 0.000,C 90.000,E1 271.661} C_DIS
LIN {X 0.214,Y -604.817,Z 972.307,A 0.000,B 0.000,C 90.000,E1 271.260} C_DIS
LIN {X 0.219,Y -598.008,Z 972.305,A 0.000,B 0.000,C 90.000,E1 270.917} C_DIS
LIN {X 0.014,Y -590.766,Z 972.304,A 0.000,B 0.000,C 90.000,E1 270.630} C_DIS
LIN {X 0.268,Y -585.381,Z 972.302,A 0.000,B 0.000,C 90.000,E1 270.401} C_DIS
LIN {X 0.194,Y -577.839,Z 972.301,A 0.000,B 0.000,C 90.000,E1 270.172} C_DIS
LIN {X -0.198,Y -572.232,Z 972.300,A 0.000,B 0.000,C 90.000,E1 270.057} C_DIS
LIN {X -0.157,Y -564.179,Z 972.299,A 0.000,B 0.000,C 90.000,E1 269.885} C_DIS
LIN {X -0.264,Y -557.343,Z 972.299,A 0.000,B 0.000,C 90.000,E1 269.828} C_DIS
LIN {X 0.235,Y -544.848,Z 972.299,A 0.000,B 0.000,C 90.000,E1 269.771} C_DIS
LIN {X -0.057,Y -543.020,Z 972.298,A 0.000,B 0.000,C 90.000,E1 269.714} C_DIS
LIN {X -0.105,Y -542.931,Z 972.298,A 0.000,B 0.000,C 90.000,E1 269.714} C_DIS
LIN {X 0.186,Y -541.289,Z 972.287,A 0.000,B 0.000,C 90.000,E1 267.593} C_DIS
LIN {X -0.175,Y -540.147,Z 972.277,A 0.000,B 0.000,C 90.000,E1 265.927} C_DIS
LIN {X -0.085,Y -539.343,Z 972.271,A 0.000,B 0.000,C 90.000,E1 264.780} C_DIS
LIN {X 0.086,Y -538.018,Z 972.261,A 0.000,B 0.000,C 90.000,E1 263.053} C_DIS
LIN {X 0.251,Y -536.968,Z 972.255,A 0.000,B 0.000,C 90.000,E1 261.894} C_DIS
LIN {X -0.013,Y -535.215,Z 972.246,A 0.000,B 0.000,C 90.000,E1 260.208} C_DIS
LIN {X 0.109,Y -533.968,Z 972.239,A 0.000,B 0.000,C 90.000,E1 259.050} C_DIS
LIN {X -0.125,Y -531.959,Z 972.230,A 0.000,B 0.000,C 90.000,E1 257.353} C_DIS
LIN {X -0.121,Y -529.509,Z 972.219,A 0.000,B 0.000,C 90.000,E1 255.338} C_DIS
LIN {X -0.190,Y -527.697,Z 972.209,A 0.000,B 0.000,C 90.000,E1 253.614} C_DIS
LIN {X 0.182,Y -526.147,Z 972.201,A 0.000,B 0.000,C 90.000,E1 252.127} C_DIS
LIN {X -0.156,Y -523.900,Z 972.191,A 0.000,B 0.000,C 90.000,E1 250.423} C_DIS
LIN {X -0.022,Y -522.010,Z 972.183,A 0.000,B 0.000,C 90.000,E1 248.954} C_DIS
LIN {X 0.072,Y -520.192,Z 972.175,A 0.000,B 0.000,C 90.000,E1 247.486} C_DIS
LIN {X 0.035,Y -518.947,Z 972.170,A 0.000,B 0.000,C 90.000,E1 246.613} C_DIS
LIN {X 0.132,Y -516.316,Z 972.160,A 0.000,B 0.000,C 90.000,E1 244.845} C_DIS
LIN {X 0.168,Y -513.583,Z 972.151,A 0.000,B 0.000,C 90.000,E1 243.076} C_DIS
LIN {X -0.182,Y -512.125,Z 972.146,A 0.000,B 0.000,C 90.000,E1 242.231} C_DIS
LIN {X -0.206,Y -510.214,Z 972.139,A 0.000,B 0.000,C 90.000,E1 241.051} C_DIS
LIN {X 0.072,Y -507.587,Z 972.131,A 0.000,B 0.000,C 90.000,E1 239.537} C_DIS
LIN {X -0.143,Y -504.682,Z 972.123,A 0.000,B 0.000,C 90.000,E1 238.074} C_DIS
LIN {X -0.059,Y -502.909,Z 972.118,A 0.000,B 0.000,C 90.000,E1 237.168} C_DIS
LIN {X 0.028,Y -500.243,Z 972.111,A 0.000,B 0.000,C 90.000,E1 235.960} C_DIS
LIN {X -0.060,Y -495.456,Z 972.099,A 0.000,B 0.000,C 90.000,E1 233.863} C_DIS
LIN {X 0.068,Y -492.721,Z 972.093,A 0.000,B 0.000,C 90.000,E1 232.637} C_DIS
LIN {X -0.003,Y -489.172,Z 972.084,A 0.000,B 0.000,C 90.000,E1 231.126} C_DIS
LIN {X -0.073,Y -484.819,Z 972.074,A 0.000,B 0.000,C 90.000,E1 229.299} C_DIS
LIN {X -0.036,Y -481.383,Z 972.065,A 0.000,B 0.000,C 90.000,E1 227.757} C_DIS
LIN {X -0.057,Y -475.975,Z 972.052,A 0.000,B 0.000,C 90.000,E1 225.283} C_DIS
LIN {X 0.126,Y -472.502,Z 972.043,A 0.000,B 0.000,C 90.000,E1 223.704} C_DIS
LIN {X 0.162,Y -469.747,Z 972.036,A 0.000,B 0.000,C 90.000,E1 222.447} C_DIS
LIN {X -0.089,Y -466.269,Z 972.027,A 0.000,B 0.000,C 90.000,E1 220.906} C_DIS
LIN {X -0.058,Y -462.718,Z 972.018,A 0.000,B 0.000,C 90.000,E1 219.322} C_DIS
LIN {X -0.029,Y -459.179,Z 972.010,A 0.000,B 0.000,C 90.000,E1 217.729} C_DIS
LIN {X 0.030,Y -454.954,Z 971.999,A 0.000,B 0.000,C 90.000,E1 215.804} C_DIS
LIN {X -0.188,Y -450.010,Z 971.986,A 0.000,B 0.000,C 90.000,E1 213.579} C_DIS
LIN {X 0.204,Y -445.064,Z 971.974,A 0.000,B 0.000,C 90.000,E1 211.258} C_DIS
LIN {X -0.107,Y -441.596,Z 971.965,A 0.000,B 0.000,C 90.000,E1 209.667} C_DIS
LIN {X -0.071,Y -437.238,Z 971.954,A 0.000,B 0.000,C 90.000,E1 207.692} C_DIS
LIN {X 0.025,Y -433.632,Z 971.945,A 0.000,B 0.000,C 90.000,E1 206.027} C_DIS
LIN {X -0.128,Y -430.594,Z 971.937,A 0.000,B 0.000,C 90.000,E1 204.719} C_DIS
LIN {X 0.007,Y -424.494,Z 971.922,A 0.000,B 0.000,C 90.000,E1 202.025} C_DIS
LIN {X 0.009,Y -418.708,Z 971.907,A 0.000,B 0.000,C 90.000,E1 199.322} C_DIS
LIN {X -0.183,Y -413.249,Z 971.892,A 0.000,B 0.000,C 90.000,E1 196.622} C_DIS
LIN {X -0.125,Y -410.081,Z 971.883,A 0.000,B 0.000,C 90.000,E1 194.898} C_DIS
LIN {X -0.137,Y -406.781,Z 971.873,A 0.000,B 0.000,C 90.000,E1 193.175} C_DIS
LIN {X -0.007,Y -402.734,Z 971.862,A 0.000,B 0.000,C 90.000,E1 191.074} C_DIS
LIN {X 0.051,Y -400.127,Z 971.854,A 0.000,B 0.000,C 90.000,E1 189.670} C_DIS
LIN {X -0.109,Y -396.108,Z 971.842,A 0.000,B 0.000,C 90.000,E1 187.587} C_DIS
LIN {X -0.061,Y -392.096,Z 971.828,A 0.000,B 0.000,C 90.000,E1 185.106} C_DIS
LIN {X 0.137,Y -390.900,Z 971.822,A 0.000,B 0.000,C 90.000,E1 184.012} C_DIS
LIN {X 0.051,Y -390.762,Z 971.820,A 0.000,B 0.000,C 90.000,E1 183.669} C_DIS
LIN {X -0.036,Y -390.488,Z 971.818,A 0.000,B 0.000,C 90.000,E1 183.326} C_DIS
LIN {X -0.187,Y -390.588,Z 971.815,A 0.000,B 0.000,C 90.000,E1 182.636} C_DIS
LIN {X 0.160,Y -390.544,Z 971.814,A 0.000,B 0.000,C 90.000,E1 182.407} C_DIS
LIN {X -0.007,Y -391.334,Z 971.810,A 0.000,B 0.000,C 90.000,E1 181.776} C_DIS
LIN {X -0.172,Y -393.308,Z 971.806,A 0.000,B 0.000,C 90.000,E1 181.088} C_DIS
LIN {X 0.109,Y -395.455,Z 971.803,A 0.000,B 0.000,C 90.000,E1 180.516} C_DIS
LIN {X 0.007,Y -400.155,Z 971.799,A 0.000,B 0.000,C 90.000,E1 179.771} C_DIS
LIN {X 0.093,Y -405.784,Z 971.795,A 0.000,B 0.000,C 90.000,E1 179.083} C_DIS
LIN {X 0.047,Y -414.572,Z 971.790,A 0.000,B 0.000,C 90.000,E1 178.224} C_DIS
LIN {X -0.135,Y -424.919,Z 971.785,A 0.000,B 0.000,C 90.000,E1 177.306} C_DIS
LIN {X -0.219,Y -435.352,Z 971.779,A 0.000,B 0.000,C 90.000,E1 176.331} C_DIS
LIN {X -0.124,Y -447.098,Z 971.773,A 0.000,B 0.000,C 90.000,E1 175.179} C_DIS
LIN {X 0.050,Y -457.222,Z 971.768,A 0.000,B 0.000,C 90.000,E1 174.147} C_DIS
LIN {X 0.233,Y -464.120,Z 971.763,A 0.000,B 0.000,C 90.000,E1 173.394} C_DIS
LIN {X 0.178,Y -470.879,Z 971.759,A 0.000,B 0.000,C 90.000,E1 172.648} C_DIS
LIN {X 0.169,Y -478.625,Z 971.754,A 0.000,B 0.000,C 90.000,E1 171.724} C_DIS
LIN {X -0.117,Y -485.935,Z 971.749,A 0.000,B 0.000,C 90.000,E1 170.849} C_DIS
LIN {X -0.117,Y -495.337,Z 971.742,A 0.000,B 0.000,C 90.000,E1 169.634} C_DIS
LIN {X -0.123,Y -502.992,Z 971.737,A 0.000,B 0.000,C 90.000,E1 168.578} C_DIS
LIN {X 0.023,Y -508.217,Z 971.732,A 0.000,B 0.000,C 90.000,E1 167.813} C_DIS
LIN {X -0.119,Y -517.004,Z 971.725,A 0.000,B 0.000,C 90.000,E1 166.520} C_DIS
LIN {X 0.165,Y -521.558,Z 971.721,A 0.000,B 0.000,C 90.000,E1 165.755} C_DIS
LIN {X 0.180,Y -531.551,Z 971.712,A 0.000,B 0.000,C 90.000,E1 164.157} C_DIS
LIN {X 0.081,Y -535.919,Z 971.708,A 0.000,B 0.000,C 90.000,E1 163.449} C_DIS
LIN {X 0.081,Y -542.620,Z 971.702,A 0.000,B 0.000,C 90.000,E1 162.308} C_DIS
LIN {X -0.214,Y -551.762,Z 971.693,A 0.000,B 0.000,C 90.000,E1 160.786} C_DIS
LIN {X 0.009,Y -558.110,Z 971.687,A 0.000,B 0.000,C 90.000,E1 159.645} C_DIS
LIN {X -0.125,Y -562.661,Z 971.682,A 0.000,B 0.000,C 90.000,E1 158.827} C_DIS
LIN {X 0.115,Y -567.151,Z 971.678,A 0.000,B 0.000,C 90.000,E1 157.975} C_DIS
LIN {X -0.131,Y -571.359,Z 971.673,A 0.000,B 0.000,C 90.000,E1 157.177} C_DIS
LIN {X 0.257,Y -576.781,Z 971.667,A 0.000,B 0.000,C 90.000,E1 156.049} C_DIS
LIN {X -0.188,Y -580.579,Z 971.663,A 0.000,B 0.000,C 90.000,E1 155.281} C_DIS
LIN {X -0.130,Y -584.669,Z 971.657,A 0.000,B 0.000,C 90.000,E1 154.332} C_DIS
LIN {X 0.027,Y -587.940,Z 971.653,A 0.000,B 0.000,C 90.000,E1 153.512} C_DIS
LIN {X -0.202,Y -590.008,Z 971.650,A 0.000,B 0.000,C 90.000,E1 152.999} C_DIS
LIN {X 0.179,Y -593.796,Z 971.644,A 0.000,B 0.000,C 90.000,E1 151.897} C_DIS
LIN {X 0.006,Y -598.040,Z 971.637,A 0.000,B 0.000,C 90.000,E1 150.589} C_DIS
LIN {X 0.131,Y -603.049,Z 971.628,A 0.000,B 0.000,C 90.000,E1 148.997} C_DIS
LIN {X 0.102,Y -608.854,Z 971.618,A 0.000,B 0.000,C 90.000,E1 147.168} C_DIS
LIN {X -0.013,Y -615.342,Z 971.606,A 0.000,B 0.000,C 90.000,E1 145.102} C_DIS
LIN {X 0.065,Y -620.949,Z 971.596,A 0.000,B 0.000,C 90.000,E1 143.290} C_DIS
LIN {X -0.355,Y -626.488,Z 971.586,A 0.000,B 0.000,C 90.000,E1 141.537} C_DIS
LIN {X 0.010,Y -630.414,Z 971.579,A 0.000,B 0.000,C 90.000,E1 140.231} C_DIS
LIN {X 0.362,Y -634.244,Z 971.572,A 0.000,B 0.000,C 90.000,E1 138.933} C_DIS
LIN {X 0.073,Y -640.535,Z 971.561,A 0.000,B 0.000,C 90.000,E1 136.944} C_DIS
LIN {X -0.023,Y -646.181,Z 971.551,A 0.000,B 0.000,C 90.000,E1 135.202} C_DIS
LIN {X -0.036,Y -652.964,Z 971.540,A 0.000,B 0.000,C 90.000,E1 133.218} C_DIS
LIN {X -0.215,Y -657.303,Z 971.533,A 0.000,B 0.000,C 90.000,E1 132.000} C_DIS
LIN {X 0.142,Y -663.723,Z 971.524,A 0.000,B 0.000,C 90.000,E1 130.253} C_DIS
LIN {X 0.156,Y -667.347,Z 971.518,A 0.000,B 0.000,C 90.000,E1 129.277} C_DIS
LIN {X -0.214,Y -671.621,Z 971.512,A 0.000,B 0.000,C 90.000,E1 128.096} C_DIS
LIN {X 0.012,Y -675.710,Z 971.505,A 0.000,B 0.000,C 90.000,E1 126.870} C_DIS
LIN {X -0.097,Y -679.461,Z 971.498,A 0.000,B 0.000,C 90.000,E1 125.678} C_DIS
LIN {X -0.142,Y -683.102,Z 971.492,A 0.000,B 0.000,C 90.000,E1 124.485} C_DIS
LIN {X -0.136,Y -686.464,Z 971.485,A 0.000,B 0.000,C 90.000,E1 123.293} C_DIS
LIN {X -0.094,Y -688.967,Z 971.480,A 0.000,B 0.000,C 90.000,E1 122.339} C_DIS
LIN {X 0.204,Y -691.931,Z 971.473,A 0.000,B 0.000,C 90.000,E1 121.131} C_DIS
LIN {X -0.042,Y -694.117,Z 971.468,A 0.000,B 0.000,C 90.000,E1 120.207} C_DIS
LIN {X -0.261,Y -695.930,Z 971.463,A 0.000,B 0.000,C 90.000,E1 119.283} C_DIS
LIN {X 0.154,Y -697.216,Z 971.457,A 0.000,B 0.000,C 90.000,E1 118.309} C_DIS
LIN {X 0.232,Y -698.411,Z 971.451,A 0.000,B 0.000,C 90.000,E1 117.129} C_DIS
LIN {X 0.093,Y -699.054,Z 971.447,A 0.000,B 0.000,C 90.000,E1 116.437} C_DIS
LIN {X -0.124,Y -699.806,Z 971.440,A 0.000,B 0.000,C 90.000,E1 115.283} C_DIS
LIN {X -0.243,Y -700.014,Z 971.437,A 0.000,B 0.000,C 90.000,E1 114.591} C_DIS
LIN {X 0.027,Y -700.047,Z 971.435,A 0.000,B 0.000,C 90.000,E1 114.335} C_DIS
LIN {X -0.360,Y -699.748,Z 971.433,A 0.000,B 0.000,C 90.000,E1 113.898} C_DIS
LIN {X -0.091,Y -699.503,Z 971.431,A 0.000,B 0.000,C 90.000,E1 113.643} C_DIS
LIN {X 0.162,Y -698.115,Z 971.429,A 0.000,B 0.000,C 90.000,E1 113.153} C_DIS
LIN {X -0.219,Y -697.185,Z 971.427,A 0.000,B 0.000,C 90.000,E1 112.950} C_DIS
LIN {X 0.038,Y -695.348,Z 971.426,A 0.000,B 0.000,C 90.000,E1 112.695} C_DIS
LIN {X 0.021,Y -693.370,Z 971.425,A 0.000,B 0.000,C 90.000,E1 112.461} C_DIS
LIN {X 0.142,Y -692.258,Z 971.424,A 0.000,B 0.000,C 90.000,E1 112.333} C_DIS
LIN {X 0.262,Y -690.752,Z 971.424,A 0.000,B 0.000,C 90.000,E1 112.206} C_DIS
LIN {X -0.361,Y -688.549,Z 971.423,A 0.000,B 0.000,C 90.000,E1 112.153} C_DIS
LIN {X -0.086,Y -686.018,Z 971.422,A 0.000,B 0.000,C 90.000,E1 112.025} C_DIS
LIN {X -0.190,Y -681.660,Z 971.422,A 0.000,B 0.000,C 90.000,E1 111.897} C_DIS
LIN {X -0.116,Y -676.837,Z 971.421,A 0.000,B 0.000,C 90.000,E1 111.770} C_DIS
LIN {X 0.133,Y -675.114,Z 971.421,A 0.000,B 0.000,C 90.000,E1 111.716} C_DIS
LIN {X -0.152,Y -667.848,Z 971.421,A 0.000,B 0.000,C 90.000,E1 111.716} C_DIS
LIN {X -0.177,Y -626.510,Z 971.421,A 0.000,B 0.000,C 90.000,E1 111.716} C_DIS
LIN {X -0.014,Y -622.663,Z 971.420,A 0.000,B 0.000,C 90.000,E1 111.642} C_DIS
LIN {X -0.167,Y -617.154,Z 971.420,A 0.000,B 0.000,C 90.000,E1 111.535} C_DIS
LIN {X 0.303,Y -610.317,Z 971.418,A 0.000,B 0.000,C 90.000,E1 111.280} C_DIS
LIN {X -0.045,Y -605.021,Z 971.417,A 0.000,B 0.000,C 90.000,E1 111.099} C_DIS
LIN {X 0.146,Y -598.368,Z 971.415,A 0.000,B 0.000,C 90.000,E1 110.737} C_DIS
LIN {X -0.130,Y -591.136,Z 971.413,A 0.000,B 0.000,C 90.000,E1 110.301} C_DIS
LIN {X 0.059,Y -584.148,Z 971.410,A 0.000,B 0.000,C 90.000,E1 109.758} C_DIS
LIN {X -0.148,Y -578.302,Z 971.407,A 0.000,B 0.000,C 90.000,E1 109.322} C_DIS
LIN {X -0.005,Y -575.423,Z 971.406,A 0.000,B 0.000,C 90.000,E1 109.087} C_DIS
LIN {X 0.062,Y -568.666,Z 971.404,A 0.000,B 0.000,C 90.000,E1 108.671} C_DIS
LIN {X -0.154,Y -567.075,Z 971.403,A 0.000,B 0.000,C 90.000,E1 108.598} C_DIS
LIN {X 0.013,Y -552.212,Z 971.399,A 0.000,B 0.000,C 90.000,E1 107.819} C_DIS
LIN {X 0.007,Y -550.159,Z 971.398,A 0.000,B 0.000,C 90.000,E1 107.638} C_DIS
LIN {X -0.030,Y -550.150,Z 971.398,A 0.000,B 0.000,C 90.000,E1 107.638} C_DIS
LIN {X -0.184,Y -549.687,Z 971.397,A 0.000,B 0.000,C 90.000,E1 107.402} C_DIS
LIN {X -0.061,Y -549.641,Z 971.394,A 0.000,B 0.000,C 90.000,E1 106.968} C_DIS
LIN {X 0.062,Y -550.258,Z 971.386,A 0.000,B 0.000,C 90.000,E1 105.552} C_DIS
LIN {X -0.278,Y -551.501,Z 971.372,A 0.000,B 0.000,C 90.000,E1 103.063} C_DIS
LIN {X -0.042,Y -554.109,Z 971.355,A 0.000,B 0.000,C 90.000,E1 99.962} C_DIS
LIN {X 0.073,Y -555.782,Z 971.346,A 0.000,B 0.000,C 90.000,E1 98.276} C_DIS
LIN {X 0.008,Y -557.069,Z 971.338,A 0.000,B 0.000,C 90.000,E1 96.891} C_DIS
LIN {X -0.091,Y -558.158,Z 971.331,A 0.000,B 0.000,C 90.000,E1 95.511} C_DIS
LIN {X -0.244,Y -558.923,Z 971.324,A 0.000,B 0.000,C 90.000,E1 94.416} C_DIS
LIN {X 0.246,Y -559.803,Z 971.317,A 0.000,B 0.000,C 90.000,E1 92.980} C_DIS
LIN {X 0.157,Y -560.532,Z 971.309,A 0.000,B 0.000,C 90.000,E1 91.604} C_DIS
LIN {X 0.167,Y -561.324,Z 971.300,A 0.000,B 0.000,C 90.000,E1 89.943} C_DIS
LIN {X 0.095,Y -561.745,Z 971.292,A 0.000,B 0.000,C 90.000,E1 88.568} C_DIS
LIN {X 0.041,Y -562.029,Z 971.284,A 0.000,B 0.000,C 90.000,E1 87.192} C_DIS
LIN {X -0.106,Y -562.249,Z 971.278,A 0.000,B 0.000,C 90.000,E1 86.102} C_DIS
LIN {X 0.025,Y -562.472,Z 971.269,A 0.000,B 0.000,C 90.000,E1 84.432} C_DIS
LIN {X 0.017,Y -562.644,Z 971.261,A 0.000,B 0.000,C 90.000,E1 83.053} C_DIS
LIN {X 0.222,Y -563.014,Z 971.252,A 0.000,B 0.000,C 90.000,E1 81.376} C_DIS
LIN {X -0.095,Y -563.918,Z 971.238,A 0.000,B 0.000,C 90.000,E1 78.926} C_DIS
LIN {X -0.041,Y -564.889,Z 971.228,A 0.000,B 0.000,C 90.000,E1 76.992} C_DIS
LIN {X 0.162,Y -566.184,Z 971.217,A 0.000,B 0.000,C 90.000,E1 75.046} C_DIS
LIN {X -0.010,Y -567.501,Z 971.206,A 0.000,B 0.000,C 90.000,E1 73.142} C_DIS
LIN {X 0.053,Y -568.402,Z 971.199,A 0.000,B 0.000,C 90.000,E1 71.764} C_DIS
LIN {X 0.115,Y -569.323,Z 971.190,A 0.000,B 0.000,C 90.000,E1 70.115} C_DIS
LIN {X 0.205,Y -570.140,Z 971.181,A 0.000,B 0.000,C 90.000,E1 68.465} C_DIS
LIN {X -0.010,Y -570.783,Z 971.171,A 0.000,B 0.000,C 90.000,E1 66.847} C_DIS
LIN {X 0.123,Y -571.129,Z 971.165,A 0.000,B 0.000,C 90.000,E1 65.741} C_DIS
LIN {X -0.200,Y -571.526,Z 971.158,A 0.000,B 0.000,C 90.000,E1 64.409} C_DIS
LIN {X 0.251,Y -571.840,Z 971.150,A 0.000,B 0.000,C 90.000,E1 62.999} C_DIS
LIN {X 0.199,Y -572.086,Z 971.143,A 0.000,B 0.000,C 90.000,E1 61.641} C_DIS
LIN {X -0.354,Y -572.203,Z 971.135,A 0.000,B 0.000,C 90.000,E1 60.333} C_DIS
LIN {X -0.004,Y -572.352,Z 971.126,A 0.000,B 0.000,C 90.000,E1 58.663} C_DIS
LIN {X -0.139,Y -572.534,Z 971.117,A 0.000,B 0.000,C 90.000,E1 57.041} C_DIS
LIN {X -0.097,Y -572.404,Z 971.109,A 0.000,B 0.000,C 90.000,E1 55.674} C_DIS
LIN {X -0.013,Y -572.351,Z 971.105,A 0.000,B 0.000,C 90.000,E1 54.848} C_DIS
LIN {X -0.263,Y -571.981,Z 971.099,A 0.000,B 0.000,C 90.000,E1 53.783} C_DIS
LIN {X 0.148,Y -571.641,Z 971.094,A 0.000,B 0.000,C 90.000,E1 52.924} C_DIS
LIN {X 0.104,Y -571.181,Z 971.090,A 0.000,B 0.000,C 90.000,E1 52.110} C_DIS
LIN {X 0.324,Y -570.208,Z 971.082,A 0.000,B 0.000,C 90.000,E1 50.723} C_DIS
LIN {X 0.081,Y -568.781,Z 971.074,A 0.000,B 0.000,C 90.000,E1 49.380} C_DIS
LIN {X 0.006,Y -567.807,Z 971.070,A 0.000,B 0.000,C 90.000,E1 48.566} C_DIS
LIN {X -0.126,Y -566.646,Z 971.065,A 0.000,B 0.000,C 90.000,E1 47.757} C_DIS
LIN {X 0.251,Y -564.822,Z 971.059,A 0.000,B 0.000,C 90.000,E1 46.620} C_DIS
LIN {X -0.223,Y -562.576,Z 971.053,A 0.000,B 0.000,C 90.000,E1 45.567} C_DIS
LIN {X -0.071,Y -561.384,Z 971.050,A 0.000,B 0.000,C 90.000,E1 45.000} C_DIS
LIN {X -0.257,Y -559.274,Z 971.045,A 0.000,B 0.000,C 90.000,E1 44.190} C_DIS
LIN {X -0.131,Y -557.739,Z 971.042,A 0.000,B 0.000,C 90.000,E1 43.623} C_DIS
LIN {X 0.047,Y -555.156,Z 971.038,A 0.000,B 0.000,C 90.000,E1 42.771} C_DIS
LIN {X 0.138,Y -553.318,Z 971.035,A 0.000,B 0.000,C 90.000,E1 42.204} C_DIS
LIN {X -0.100,Y -550.175,Z 971.030,A 0.000,B 0.000,C 90.000,E1 41.391} C_DIS
LIN {X -0.206,Y -547.262,Z 971.026,A 0.000,B 0.000,C 90.000,E1 40.701} C_DIS
LIN {X 0.077,Y -544.175,Z 971.022,A 0.000,B 0.000,C 90.000,E1 39.967} C_DIS
LIN {X -0.119,Y -542.213,Z 971.020,A 0.000,B 0.000,C 90.000,E1 39.564} C_DIS
LIN {X 0.113,Y -538.619,Z 971.016,A 0.000,B 0.000,C 90.000,E1 38.830} C_DIS
LIN {X 0.309,Y -533.235,Z 971.010,A 0.000,B 0.000,C 90.000,E1 37.810} C_DIS
LIN {X -0.306,Y -527.419,Z 971.005,A 0.000,B 0.000,C 90.000,E1 36.870} C_DIS
LIN {X 0.033,Y -522.204,Z 971.000,A 0.000,B 0.000,C 90.000,E1 35.964} C_DIS
LIN {X -0.055,Y -518.587,Z 970.997,A 0.000,B 0.000,C 90.000,E1 35.391} C_DIS
LIN {X 0.182,Y -512.813,Z 970.992,A 0.000,B 0.000,C 90.000,E1 34.485} C_DIS
LIN {X -0.167,Y -507.544,Z 970.988,A 0.000,B 0.000,C 90.000,E1 33.785} C_DIS
LIN {X -0.059,Y -500.696,Z 970.983,A 0.000,B 0.000,C 90.000,E1 32.880} C_DIS
LIN {X 0.104,Y -495.681,Z 970.979,A 0.000,B 0.000,C 90.000,E1 32.260} C_DIS
LIN {X -0.049,Y -487.625,Z 970.974,A 0.000,B 0.000,C 90.000,E1 31.386} C_DIS
LIN {X 0.141,Y -483.338,Z 970.972,A 0.000,B 0.000,C 90.000,E1 30.924} C_DIS
LIN {X 0.004,Y -473.748,Z 970.967,A 0.000,B 0.000,C 90.000,E1 30.001} C_DIS
LIN {X -0.215,Y -464.930,Z 970.962,A 0.000,B 0.000,C 90.000,E1 29.205} C_DIS
LIN {X 0.170,Y -458.935,Z 970.959,A 0.000,B 0.000,C 90.000,E1 28.615} C_DIS
LIN {X 0.067,Y -451.497,Z 970.956,A 0.000,B 0.000,C 90.000,E1 27.975} C_DIS
LIN {X 0.118,Y -436.485,Z 970.948,A 0.000,B 0.000,C 90.000,E1 26.693} C_DIS
LIN {X -0.003,Y -416.982,Z 970.939,A 0.000,B 0.000,C 90.000,E1 24.951} C_DIS
LIN {X -0.048,Y -403.857,Z 970.931,A 0.000,B 0.000,C 90.000,E1 23.643} C_DIS
LIN {X -0.239,Y -396.975,Z 970.927,A 0.000,B 0.000,C 90.000,E1 22.898} C_DIS
LIN {X -0.172,Y -393.912,Z 970.925,A 0.000,B 0.000,C 90.000,E1 22.461} C_DIS
LIN {X 0.036,Y -393.032,Z 970.924,A 0.000,B 0.000,C 90.000,E1 22.280} C_DIS
LIN {X -0.095,Y -391.808,Z 970.922,A 0.000,B 0.000,C 90.000,E1 21.972} C_DIS
LIN {X -0.016,Y -390.748,Z 970.921,A 0.000,B 0.000,C 90.000,E1 21.716} C_DIS
LIN {X 0.139,Y -390.024,Z 970.918,A 0.000,B 0.000,C 90.000,E1 21.227} C_DIS
LIN {X -0.219,Y -389.828,Z 970.916,A 0.000,B 0.000,C 90.000,E1 20.918} C_DIS
LIN {X -0.179,Y -389.783,Z 970.914,A 0.000,B 0.000,C 90.000,E1 20.556} C_DIS
LIN {X 0.074,Y -390.325,Z 970.908,A 0.000,B 0.000,C 90.000,E1 19.450} C_DIS
LIN {X -0.099,Y -392.681,Z 970.894,A 0.000,B 0.000,C 90.000,E1 16.985} C_DIS
LIN {X 0.082,Y -396.440,Z 970.877,A 0.000,B 0.000,C 90.000,E1 13.772} C_DIS
LIN {X 0.153,Y -399.889,Z 970.863,A 0.000,B 0.000,C 90.000,E1 11.299} C_DIS
LIN {X 0.087,Y -405.123,Z 970.845,A 0.000,B 0.000,C 90.000,E1 8.163} C_DIS
LIN {X 0.059,Y -411.024,Z 970.828,A 0.000,B 0.000,C 90.000,E1 5.049} C_DIS
LIN {X 0.120,Y -415.408,Z 970.817,A 0.000,B 0.000,C 90.000,E1 2.980} C_DIS
LIN {X -0.147,Y -420.944,Z 970.803,A 0.000,B 0.000,C 90.000,E1 0.630} C_DIS
LIN {X 0.000,Y -422.772,Z 970.800,A 0.000,B 0.000,C 90.000,E1 360.000} C_DIS
LIN {X 0.086,Y -425.582,Z 970.797,A 0.000,B 0.000,C 90.000,E1 359.370} C_DIS
LIN {X 0.167,Y -429.144,Z 970.794,A 0.000,B 0.000,C 90.000,E1 358.854} C_DIS
LIN {X 0.052,Y -430.438,Z 970.793,A 0.000,B 0.000,C 90.000,E1 358.740} C_DIS
LIN {X -0.179,Y -433.575,Z 970.792,A 0.000,B 0.000,C 90.000,E1 358.511} C_DIS
LIN {X -0.004,Y -437.719,Z 970.790,A 0.000,B 0.000,C 90.000,E1 358.224} C_DIS
LIN {X -0.190,Y -441.041,Z 970.789,A 0.000,B 0.000,C 90.000,E1 358.051} C_DIS
LIN {X -0.222,Y -450.762,Z 970.786,A 0.000,B 0.000,C 90.000,E1 357.535} C_DIS
LIN {X -0.199,Y -467.570,Z 970.781,A 0.000,B 0.000,C 90.000,E1 356.617} C_DIS
LIN {X 0.105,Y -474.391,Z 970.779,A 0.000,B 0.000,C 90.000,E1 356.216} C_DIS
LIN {X -0.140,Y -489.198,Z 970.774,A 0.000,B 0.000,C 90.000,E1 355.412} C_DIS
LIN {X 0.088,Y -503.714,Z 970.770,A 0.000,B 0.000,C 90.000,E1 354.546} C_DIS
LIN {X 0.244,Y -509.991,Z 970.768,A 0.000,B 0.000,C 90.000,E1 354.147} C_DIS
LIN {X -0.146,Y -519.419,Z 970.764,A 0.000,B 0.000,C 90.000,E1 353.571} C_DIS
LIN {X -0.281,Y -527.172,Z 970.761,A 0.000,B 0.000,C 90.000,E1 353.053} C_DIS
LIN {X -0.079,Y -534.533,Z 970.758,A 0.000,B 0.000,C 90.000,E1 352.470} C_DIS
LIN {X -0.268,Y -541.626,Z 970.755,A 0.000,B 0.000,C 90.000,E1 351.894} C_DIS
LIN {X -0.118,Y -547.096,Z 970.752,A 0.000,B 0.000,C 90.000,E1 351.376} C_DIS
LIN {X 0.110,Y -554.844,Z 970.748,A 0.000,B 0.000,C 90.000,E1 350.557} C_DIS
LIN {X 0.033,Y -558.638,Z 970.745,A 0.000,B 0.000,C 90.000,E1 350.151} C_DIS
LIN {X -0.122,Y -565.141,Z 970.741,A 0.000,B 0.000,C 90.000,E1 349.342} C_DIS
LIN {X 0.214,Y -569.227,Z 970.738,A 0.000,B 0.000,C 90.000,E1 348.757} C_DIS
LIN {X 0.023,Y -573.060,Z 970.735,A 0.000,B 0.000,C 90.000,E1 348.229} C_DIS
LIN {X 0.308,Y -577.425,Z 970.731,A 0.000,B 0.000,C 90.000,E1 347.521} C_DIS
LIN {X -0.165,Y -582.299,Z 970.726,A 0.000,B 0.000,C 90.000,E1 346.756} C_DIS
LIN {X -0.025,Y -586.753,Z 970.722,A 0.000,B 0.000,C 90.000,E1 345.936} C_DIS
LIN {X -0.004,Y -592.385,Z 970.716,A 0.000,B 0.000,C 90.000,E1 344.866} C_DIS
LIN {X -0.345,Y -596.336,Z 970.712,A 0.000,B 0.000,C 90.000,E1 344.102} C_DIS
LIN {X 0.088,Y -600.210,Z 970.707,A 0.000,B 0.000,C 90.000,E1 343.268} C_DIS
LIN {X -0.063,Y -604.407,Z 970.702,A 0.000,B 0.000,C 90.000,E1 342.362} C_DIS
LIN {X -0.204,Y -608.843,Z 970.696,A 0.000,B 0.000,C 90.000,E1 341.329} C_DIS
LIN {X 0.035,Y -614.161,Z 970.689,A 0.000,B 0.000,C 90.000,E1 340.007} C_DIS
LIN {X 0.273,Y -617.102,Z 970.685,A 0.000,B 0.000,C 90.000,E1 339.209} C_DIS
LIN {X -0.033,Y -619.808,Z 970.680,A 0.000,B 0.000,C 90.000,E1 338.465} C_DIS
LIN {X 0.259,Y -623.338,Z 970.675,A 0.000,B 0.000,C 90.000,E1 337.411} C_DIS
LIN {X 0.026,Y -626.571,Z 970.669,A 0.000,B 0.000,C 90.000,E1 336.410} C_DIS
LIN {X -0.186,Y -628.997,Z 970.665,A 0.000,B 0.000,C 90.000,E1 335.665} C_DIS
LIN {X -0.354,Y -631.889,Z 970.659,A 0.000,B 0.000,C 90.000,E1 334.665} C_DIS
LIN {X -0.253,Y -633.951,Z 970.655,A 0.000,B 0.000,C 90.000,E1 333.896} C_DIS
LIN {X 0.013,Y -637.647,Z 970.646,A 0.000,B 0.000,C 90.000,E1 332.359} C_DIS
LIN {X 0.089,Y -640.953,Z 970.638,A 0.000,B 0.000,C 90.000,E1 330.845} C_DIS
LIN {X -0.219,Y -643.003,Z 970.633,A 0.000,B 0.000,C 90.000,E1 329.871} C_DIS
LIN {X -0.183,Y -644.889,Z 970.627,A 0.000,B 0.000,C 90.000,E1 328.869} C_DIS
LIN {X -0.122,Y -646.483,Z 970.621,A 0.000,B 0.000,C 90.000,E1 327.867} C_DIS
LIN {X 0.306,Y -647.971,Z 970.616,A 0.000,B 0.000,C 90.000,E1 326.834} C_DIS
LIN {X -0.143,Y -649.228,Z 970.610,A 0.000,B 0.000,C 90.000,E1 325.881} C_DIS
LIN {X 0.227,Y -650.536,Z 970.604,A 0.000,B 0.000,C 90.000,E1 324.609} C_DIS
LIN {X -0.288,Y -651.617,Z 970.597,A 0.000,B 0.000,C 90.000,E1 323.417} C_DIS
LIN {X 0.114,Y -652.476,Z 970.590,A 0.000,B 0.000,C 90.000,E1 322.145} C_DIS
LIN {X -0.035,Y -653.049,Z 970.584,A 0.000,B 0.000,C 90.000,E1 321.170} C_DIS
LIN {X -0.166,Y -653.526,Z 970.579,A 0.000,B 0.000,C 90.000,E1 320.194} C_DIS
LIN {X 0.111,Y -654.251,Z 970.571,A 0.000,B 0.000,C 90.000,E1 318.690} C_DIS
LIN {X 0.201,Y -656.167,Z 970.556,A 0.000,B 0.000,C 90.000,E1 315.972} C_DIS
LIN {X 0.102,Y -656.767,Z 970.551,A 0.000,B 0.000,C 90.000,E1 315.243} C_DIS
LIN {X -0.167,Y -658.546,Z 970.539,A 0.000,B 0.000,C 90.000,E1 313.056} C_DIS
LIN {X -0.293,Y -659.807,Z 970.531,A 0.000,B 0.000,C 90.000,E1 311.595} C_DIS
LIN {X 0.107,Y -660.855,Z 970.523,A 0.000,B 0.000,C 90.000,E1 310.092} C_DIS
LIN {X -0.374,Y -661.646,Z 970.516,A 0.000,B 0.000,C 90.000,E1 308.910} C_DIS
LIN {X 0.084,Y -662.319,Z 970.509,A 0.000,B 0.000,C 90.000,E1 307.649} C_DIS
LIN {X -0.307,Y -662.681,Z 970.505,A 0.000,B 0.000,C 90.000,E1 306.950} C_DIS
LIN {X 0.245,Y -663.040,Z 970.497,A 0.000,B 0.000,C 90.000,E1 305.438} C_DIS
LIN {X 0.212,Y -663.609,Z 970.485,A 0.000,B 0.000,C 90.000,E1 303.245} C_DIS
LIN {X -0.099,Y -665.801,Z 970.465,A 0.000,B 0.000,C 90.000,E1 299.617} C_DIS
LIN {X 0.068,Y -671.159,Z 970.443,A 0.000,B 0.000,C 90.000,E1 295.720} C_DIS
LIN {X 0.097,Y -674.185,Z 970.434,A 0.000,B 0.000,C 90.000,E1 294.027} C_DIS
LIN {X -0.082,Y -675.729,Z 970.428,A 0.000,B 0.000,C 90.000,E1 293.078} C_DIS
LIN {X 0.096,Y -676.059,Z 970.427,A 0.000,B 0.000,C 90.000,E1 292.823} C_DIS
LIN {X 0.193,Y -676.361,Z 970.424,A 0.000,B 0.000,C 90.000,E1 292.333} C_DIS
LIN {X 0.117,Y -676.358,Z 970.423,A 0.000,B 0.000,C 90.000,E1 292.099} C_DIS
LIN {X -0.155,Y -675.908,Z 970.420,A 0.000,B 0.000,C 90.000,E1 291.642} C_DIS
LIN {X -0.228,Y -675.300,Z 970.419,A 0.000,B 0.000,C 90.000,E1 291.408} C_DIS
LIN {X -0.055,Y -674.476,Z 970.418,A 0.000,B 0.000,C 90.000,E1 291.153} C_DIS
LIN {X -0.127,Y -673.344,Z 970.416,A 0.000,B 0.000,C 90.000,E1 290.918} C_DIS
LIN {X -0.044,Y -672.640,Z 970.416,A 0.000,B 0.000,C 90.000,E1 290.791} C_DIS
LIN {X 0.038,Y -671.603,Z 970.415,A 0.000,B 0.000,C 90.000,E1 290.663} C_DIS
LIN {X -0.091,Y -666.380,Z 970.412,A 0.000,B 0.000,C 90.000,E1 290.248} C_DIS
LIN {X 0.116,Y -664.867,Z 970.412,A 0.000,B 0.000,C 90.000,E1 290.120} C_DIS
LIN {X 0.042,Y -655.252,Z 970.409,A 0.000,B 0.000,C 90.000,E1 289.523} C_DIS
LIN {X 0.194,Y -655.184,Z 970.409,A 0.000,B 0.000,C 90.000,E1 289.504} C_DIS
LIN {X -0.123,Y -653.621,Z 970.407,A 0.000,B 0.000,C 90.000,E1 289.322} C_DIS
LIN {X -0.167,Y -653.592,Z 970.407,A 0.000,B 0.000,C 90.000,E1 289.322} C_DIS
LIN {X 0.056,Y -653.920,Z 970.406,A 0.000,B 0.000,C 90.000,E1 289.087} C_DIS
LIN {X -0.030,Y -655.339,Z 970.404,A 0.000,B 0.000,C 90.000,E1 288.725} C_DIS
LIN {X -0.069,Y -658.136,Z 970.401,A 0.000,B 0.000,C 90.000,E1 288.236} C_DIS
LIN {X -0.346,Y -663.315,Z 970.397,A 0.000,B 0.000,C 90.000,E1 287.402} C_DIS
LIN {X 0.351,Y -666.599,Z 970.393,A 0.000,B 0.000,C 90.000,E1 286.732} C_DIS
LIN {X 0.186,Y -668.853,Z 970.391,A 0.000,B 0.000,C 90.000,E1 286.260} C_DIS
LIN {X 0.109,Y -669.904,Z 970.389,A 0.000,B 0.000,C 90.000,E1 286.024} C_DIS
LIN {X 0.080,Y -672.352,Z 970.385,A 0.000,B 0.000,C 90.000,E1 285.300} C_DIS
LIN {X -0.048,Y -673.672,Z 970.382,A 0.000,B 0.000,C 90.000,E1 284.828} C_DIS
LIN {X -0.221,Y -675.178,Z 970.378,A 0.000,B 0.000,C 90.000,E1 284.120} C_DIS
LIN {X 0.330,Y -675.959,Z 970.376,A 0.000,B 0.000,C 90.000,E1 283.592} C_DIS
LIN {X 0.179,Y -676.821,Z 970.372,A 0.000,B 0.000,C 90.000,E1 282.883} C_DIS
LIN {X -0.109,Y -677.383,Z 970.368,A 0.000,B 0.000,C 90.000,E1 282.187} C_DIS
LIN {X -0.155,Y -677.526,Z 970.366,A 0.000,B 0.000,C 90.000,E1 281.951} C_DIS
LIN {X -0.296,Y -677.522,Z 970.362,A 0.000,B 0.000,C 90.000,E1 281.243} C_DIS
LIN {X 0.144,Y -677.270,Z 970.360,A 0.000,B 0.000,C 90.000,E1 280.725} C_DIS
LIN {X 0.045,Y -676.753,Z 970.357,A 0.000,B 0.000,C 90.000,E1 280.254} C_DIS
LIN {X -0.178,Y -675.967,Z 970.354,A 0.000,B 0.000,C 90.000,E1 279.792} C_DIS
LIN {X 0.313,Y -674.326,Z 970.350,A 0.000,B 0.000,C 90.000,E1 279.029} C_DIS
LIN {X 0.077,Y -672.857,Z 970.348,A 0.000,B 0.000,C 90.000,E1 278.568} C_DIS
LIN {X -0.241,Y -670.051,Z 970.344,A 0.000,B 0.000,C 90.000,E1 277.871} C_DIS
LIN {X 0.250,Y -669.027,Z 970.342,A 0.000,B 0.000,C 90.000,E1 277.587} C_DIS
LIN {X -0.019,Y -665.962,Z 970.339,A 0.000,B 0.000,C 90.000,E1 277.004} C_DIS
LIN {X 0.262,Y -662.339,Z 970.336,A 0.000,B 0.000,C 90.000,E1 276.372} C_DIS
LIN {X -0.046,Y -658.997,Z 970.333,A 0.000,B 0.000,C 90.000,E1 275.910} C_DIS
LIN {X 0.175,Y -654.165,Z 970.329,A 0.000,B 0.000,C 90.000,E1 275.277} C_DIS
LIN {X -0.291,Y -648.804,Z 970.326,A 0.000,B 0.000,C 90.000,E1 274.702} C_DIS
LIN {X 0.024,Y -645.390,Z 970.324,A 0.000,B 0.000,C 90.000,E1 274.302} C_DIS
LIN {X -0.242,Y -639.353,Z 970.321,A 0.000,B 0.000,C 90.000,E1 273.726} C_DIS
LIN {X 0.182,Y -632.739,Z 970.317,A 0.000,B 0.000,C 90.000,E1 273.094} C_DIS
LIN {X 0.245,Y -625.691,Z 970.314,A 0.000,B 0.000,C 90.000,E1 272.522} C_DIS
LIN {X 0.083,Y -618.436,Z 970.311,A 0.000,B 0.000,C 90.000,E1 272.007} C_DIS
LIN {X -0.282,Y -610.661,Z 970.308,A 0.000,B 0.000,C 90.000,E1 271.547} C_DIS
LIN {X 0.044,Y -604.151,Z 970.306,A 0.000,B 0.000,C 90.000,E1 271.146} C_DIS
LIN {X 0.096,Y -597.279,Z 970.305,A 0.000,B 0.000,C 90.000,E1 270.802} C_DIS
LIN {X -0.022,Y -590.080,Z 970.303,A 0.000,B 0.000,C 90.000,E1 270.516} C_DIS
LIN {X 0.273,Y -584.784,Z 970.302,A 0.000,B 0.000,C 90.000,E1 270.286} C_DIS
LIN {X 0.252,Y -577.323,Z 970.301,A 0.000,B 0.000,C 90.000,E1 270.057} C_DIS
LIN {X -0.126,Y -571.549,Z 970.300,A 0.000,B 0.000,C 90.000,E1 269.943} C_DIS
LIN {X -0.275,Y -565.363,Z 970.299,A 0.000,B 0.000,C 90.000,E1 269.828} C_DIS
LIN {X -0.070,Y -557.395,Z 970.298,A 0.000,B 0.000,C 90.000,E1 269.714} C_DIS
LIN {X -0.124,Y -546.296,Z 970.298,A 0.000,B 0.000,C 90.000,E1 269.714} C_DIS
LIN {X -0.028,Y -542.971,Z 970.297,A 0.000,B 0.000,C 90.000,E1 269.542} C_DIS
LIN {X -0.077,Y -542.927,Z 970.297,A 0.000,B 0.000,C 90.000,E1 269.542} C_DIS
LIN {X -0.160,Y -541.295,Z 970.286,A 0.000,B 0.000,C 90.000,E1 267.535} C_DIS
LIN {X 0.019,Y -540.172,Z 970.277,A 0.000,B 0.000,C 90.000,E1 265.812} C_DIS
LIN {X 0.106,Y -539.363,Z 970.270,A 0.000,B 0.000,C 90.000,E1 264.666} C_DIS
LIN {X -0.194,Y -538.058,Z 970.261,A 0.000,B 0.000,C 90.000,E1 262.989} C_DIS
LIN {X -0.036,Y -536.717,Z 970.253,A 0.000,B 0.000,C 90.000,E1 261.546} C_DIS
LIN {X 0.224,Y -534.959,Z 970.244,A 0.000,B 0.000,C 90.000,E1 259.803} C_DIS
LIN {X -0.188,Y -533.607,Z 970.237,A 0.000,B 0.000,C 90.000,E1 258.701} C_DIS
LIN {X 0.160,Y -531.935,Z 970.229,A 0.000,B 0.000,C 90.000,E1 257.229} C_DIS
LIN {X 0.006,Y -529.837,Z 970.220,A 0.000,B 0.000,C 90.000,E1 255.519} C_DIS
LIN {X -0.041,Y -527.680,Z 970.208,A 0.000,B 0.000,C 90.000,E1 253.504} C_DIS
LIN {X -0.016,Y -526.099,Z 970.200,A 0.000,B 0.000,C 90.000,E1 252.054} C_DIS
LIN {X -0.027,Y -523.859,Z 970.191,A 0.000,B 0.000,C 90.000,E1 250.315} C_DIS
LIN {X -0.059,Y -522.373,Z 970.184,A 0.000,B 0.000,C 90.000,E1 249.156} C_DIS
LIN {X -0.101,Y -520.141,Z 970.174,A 0.000,B 0.000,C 90.000,E1 247.411} C_DIS
LIN {X 0.010,Y -518.425,Z 970.168,A 0.000,B 0.000,C 90.000,E1 246.230} C_DIS
LIN {X -0.248,Y -516.231,Z 970.160,A 0.000,B 0.000,C 90.000,E1 244.793} C_DIS
LIN {X -0.104,Y -513.949,Z 970.152,A 0.000,B 0.000,C 90.000,E1 243.307} C_DIS
LIN {X 0.012,Y -512.552,Z 970.147,A 0.000,B 0.000,C 90.000,E1 242.410} C_DIS
LIN {X 0.092,Y -510.111,Z 970.139,A 0.000,B 0.000,C 90.000,E1 240.923} C_DIS
LIN {X 0.037,Y -508.010,Z 970.132,A 0.000,B 0.000,C 90.000,E1 239.744} C_DIS
LIN {X 0.205,Y -505.746,Z 970.125,A 0.000,B 0.000,C 90.000,E1 238.535} C_DIS
LIN {X -0.085,Y -503.409,Z 970.119,A 0.000,B 0.000,C 90.000,E1 237.375} C_DIS
LIN {X 0.011,Y -500.760,Z 970.112,A 0.000,B 0.000,C 90.000,E1 236.167} C_DIS
LIN {X -0.203,Y -497.308,Z 970.104,A 0.000,B 0.000,C 90.000,E1 234.689} C_DIS
LIN {X 0.075,Y -493.293,Z 970.094,A 0.000,B 0.000,C 90.000,E1 232.844} C_DIS
LIN {X 0.167,Y -489.009,Z 970.084,A 0.000,B 0.000,C 90.000,E1 231.009} C_DIS
LIN {X 0.294,Y -483.991,Z 970.072,A 0.000,B 0.000,C 90.000,E1 228.852} C_DIS
LIN {X 0.183,Y -481.233,Z 970.065,A 0.000,B 0.000,C 90.000,E1 227.634} C_DIS
LIN {X 0.137,Y -475.829,Z 970.051,A 0.000,B 0.000,C 90.000,E1 225.162} C_DIS
LIN {X -0.016,Y -472.351,Z 970.042,A 0.000,B 0.000,C 90.000,E1 223.623} C_DIS
LIN {X -0.066,Y -470.307,Z 970.037,A 0.000,B 0.000,C 90.000,E1 222.690} C_DIS
LIN {X 0.118,Y -466.112,Z 970.027,A 0.000,B 0.000,C 90.000,E1 220.782} C_DIS
LIN {X 0.151,Y -462.591,Z 970.018,A 0.000,B 0.000,C 90.000,E1 219.197} C_DIS
LIN {X -0.077,Y -458.346,Z 970.007,A 0.000,B 0.000,C 90.000,E1 217.317} C_DIS
LIN {X -0.031,Y -454.092,Z 969.997,A 0.000,B 0.000,C 90.000,E1 215.391} C_DIS
LIN {X 0.023,Y -449.861,Z 969.986,A 0.000,B 0.000,C 90.000,E1 213.452} C_DIS
LIN {X -0.034,Y -445.634,Z 969.975,A 0.000,B 0.000,C 90.000,E1 211.514} C_DIS
LIN {X 0.046,Y -442.150,Z 969.966,A 0.000,B 0.000,C 90.000,E1 209.873} C_DIS
LIN {X 0.064,Y -438.516,Z 969.957,A 0.000,B 0.000,C 90.000,E1 208.231} C_DIS
LIN {X 0.209,Y -434.217,Z 969.946,A 0.000,B 0.000,C 90.000,E1 206.232} C_DIS
LIN {X 0.064,Y -430.450,Z 969.937,A 0.000,B 0.000,C 90.000,E1 204.591} C_DIS
LIN {X 0.188,Y -424.303,Z 969.922,A 0.000,B 0.000,C 90.000,E1 201.897} C_DIS
LIN {X -0.129,Y -419.282,Z 969.909,A 0.000,B 0.000,C 90.000,E1 199.577} C_DIS
LIN {X -0.169,Y -413.776,Z 969.894,A 0.000,B 0.000,C 90.000,E1 196.858} C_DIS
LIN {X 0.024,Y -409.918,Z 969.882,A 0.000,B 0.000,C 90.000,E1 194.773} C_DIS
LIN {X -0.092,Y -406.570,Z 969.873,A 0.000,B 0.000,C 90.000,E1 193.063} C_DIS
LIN {X 0.117,Y -403.204,Z 969.863,A 0.000,B 0.000,C 90.000,E1 191.299} C_DIS
LIN {X 0.098,Y -399.920,Z 969.853,A 0.000,B 0.000,C 90.000,E1 189.557} C_DIS
LIN {X 0.014,Y -396.553,Z 969.843,A 0.000,B 0.000,C 90.000,E1 187.814} C_DIS
LIN {X -0.070,Y -391.264,Z 969.826,A 0.000,B 0.000,C 90.000,E1 184.645} C_DIS
LIN {X 0.045,Y -390.105,Z 969.819,A 0.000,B 0.000,C 90.000,E1 183.383} C_DIS
LIN {X 0.137,Y -389.983,Z 969.813,A 0.000,B 0.000,C 90.000,E1 182.236} C_DIS
LIN {X 0.050,Y -390.274,Z 969.811,A 0.000,B 0.000,C 90.000,E1 181.892} C_DIS
LIN {X -0.068,Y -391.107,Z 969.808,A 0.000,B 0.000,C 90.000,E1 181.375} C_DIS
LIN {X -0.193,Y -392.588,Z 969.805,A 0.000,B 0.000,C 90.000,E1 180.859} C_DIS
LIN {X 0.120,Y -394.672,Z 969.802,A 0.000,B 0.000,C 90.000,E1 180.286} C_DIS
LIN {X 0.057,Y -399.156,Z 969.798,A 0.000,B 0.000,C 90.000,E1 179.542} C_DIS
LIN {X 0.062,Y -404.803,Z 969.794,A 0.000,B 0.000,C 90.000,E1 178.854} C_DIS
LIN {X -0.172,Y -412.619,Z 969.789,A 0.000,B 0.000,C 90.000,E1 178.108} C_DIS
LIN {X -0.137,Y -423.333,Z 969.784,A 0.000,B 0.000,C 90.000,E1 177.135} C_DIS
LIN {X 0.022,Y -432.333,Z 969.779,A 0.000,B 0.000,C 90.000,E1 176.274} C_DIS
LIN {X -0.043,Y -445.717,Z 969.772,A 0.000,B 0.000,C 90.000,E1 175.008} C_DIS
LIN {X -0.033,Y -455.554,Z 969.767,A 0.000,B 0.000,C 90.000,E1 174.033} C_DIS
LIN {X -0.012,Y -461.161,Z 969.764,A 0.000,B 0.000,C 90.000,E1 173.451} C_DIS
LIN {X -0.137,Y -466.632,Z 969.760,A 0.000,B 0.000,C 90.000,E1 172.875} C_DIS
LIN {X 0.058,Y -472.039,Z 969.757,A 0.000,B 0.000,C 90.000,E1 172.243} C_DIS
LIN {X 0.237,Y -480.991,Z 969.751,A 0.000,B 0.000,C 90.000,E1 171.141} C_DIS
LIN {X -0.040,Y -489.518,Z 969.745,A 0.000,B 0.000,C 90.000,E1 170.095} C_DIS
LIN {X -0.116,Y -495.402,Z 969.741,A 0.000,B 0.000,C 90.000,E1 169.342} C_DIS
LIN {X 0.111,Y -501.980,Z 969.736,A 0.000,B 0.000,C 90.000,E1 168.409} C_DIS
LIN {X -0.249,Y -507.300,Z 969.732,A 0.000,B 0.000,C 90.000,E1 167.701} C_DIS
LIN {X 0.150,Y -511.269,Z 969.728,A 0.000,B 0.000,C 90.000,E1 167.061} C_DIS
LIN {X -0.001,Y -514.404,Z 969.726,A 0.000,B 0.000,C 90.000,E1 166.645} C_DIS
LIN {X -0.263,Y -520.796,Z 969.720,A 0.000,B 0.000,C 90.000,E1 165.644} C_DIS
LIN {X 0.038,Y -529.944,Z 969.712,A 0.000,B 0.000,C 90.000,E1 164.157} C_DIS
LIN {X 0.115,Y -536.097,Z 969.706,A 0.000,B 0.000,C 90.000,E1 163.142} C_DIS
LIN {X -0.248,Y -541.972,Z 969.701,A 0.000,B 0.000,C 90.000,E1 162.181} C_DIS
LIN {X 0.094,Y -550.353,Z 969.693,A 0.000,B 0.000,C 90.000,E1 160.732} C_DIS
LIN {X -0.033,Y -556.765,Z 969.687,A 0.000,B 0.000,C 90.000,E1 159.625} C_DIS
LIN {X -0.064,Y -562.897,Z 969.681,A 0.000,B 0.000,C 90.000,E1 158.518} C_DIS
LIN {X 0.177,Y -567.336,Z 969.676,A 0.000,B 0.000,C 90.000,E1 157.667} C_DIS
LIN {X -0.241,Y -572.941,Z 969.670,A 0.000,B 0.000,C 90.000,E1 156.613} C_DIS
LIN {X 0.096,Y -578.911,Z 969.663,A 0.000,B 0.000,C 90.000,E1 155.357} C_DIS
LIN {X 0.267,Y -581.937,Z 969.659,A 0.000,B 0.000,C 90.000,E1 154.665} C_DIS
LIN {X -0.129,Y -585.285,Z 969.655,A 0.000,B 0.000,C 90.000,E1 153.896} C_DIS
LIN {X 0.030,Y -588.501,Z 969.651,A 0.000,B 0.000,C 90.000,E1 153.076} C_DIS
LIN {X -0.138,Y -592.407,Z 969.645,A 0.000,B 0.000,C 90.000,E1 152.025} C_DIS
LIN {X 0.278,Y -595.935,Z 969.639,A 0.000,B 0.000,C 90.000,E1 150.923} C_DIS
LIN {X 0.136,Y -600.169,Z 969.631,A 0.000,B 0.000,C 90.000,E1 149.616} C_DIS
LIN {X -0.148,Y -604.383,Z 969.624,A 0.000,B 0.000,C 90.000,E1 148.329} C_DIS
LIN {X 0.152,Y -608.553,Z 969.617,A 0.000,B 0.000,C 90.000,E1 146.993} C_DIS
LIN {X 0.069,Y -614.285,Z 969.607,A 0.000,B 0.000,C 90.000,E1 145.182} C_DIS
LIN {X -0.377,Y -619.944,Z 969.597,A 0.000,B 0.000,C 90.000,E1 143.417} C_DIS
LIN {X -0.326,Y -625.526,Z 969.587,A 0.000,B 0.000,C 90.000,E1 141.618} C_DIS
LIN {X 0.071,Y -628.728,Z 969.581,A 0.000,B 0.000,C 90.000,E1 140.561} C_DIS
LIN {X -0.124,Y -633.383,Z 969.573,A 0.000,B 0.000,C 90.000,E1 139.057} C_DIS
LIN {X -0.050,Y -640.589,Z 969.560,A 0.000,B 0.000,C 90.000,E1 136.782} C_DIS
LIN {X 0.246,Y -647.159,Z 969.549,A 0.000,B 0.000,C 90.000,E1 134.757} C_DIS
LIN {X -0.155,Y -653.162,Z 969.539,A 0.000,B 0.000,C 90.000,E1 133.056} C_DIS
LIN {X 0.060,Y -660.275,Z 969.528,A 0.000,B 0.000,C 90.000,E1 131.067} C_DIS
LIN {X 0.004,Y -664.899,Z 969.521,A 0.000,B 0.000,C 90.000,E1 129.850} C_DIS
LIN {X 0.024,Y -668.503,Z 969.516,A 0.000,B 0.000,C 90.000,E1 128.874} C_DIS
LIN {X 0.198,Y -671.869,Z 969.511,A 0.000,B 0.000,C 90.000,E1 127.890} C_DIS
LIN {X -0.104,Y -675.252,Z 969.505,A 0.000,B 0.000,C 90.000,E1 126.950} C_DIS
LIN {X 0.179,Y -679.036,Z 969.499,A 0.000,B 0.000,C 90.000,E1 125.724} C_DIS
LIN {X 0.121,Y -682.701,Z 969.492,A 0.000,B 0.000,C 90.000,E1 124.532} C_DIS
LIN {X -0.263,Y -686.076,Z 969.485,A 0.000,B 0.000,C 90.000,E1 123.372} C_DIS
LIN {X -0.224,Y -688.620,Z 969.480,A 0.000,B 0.000,C 90.000,E1 122.418} C_DIS
LIN {X -0.290,Y -692.150,Z 969.472,A 0.000,B 0.000,C 90.000,E1 121.003} C_DIS
LIN {X -0.186,Y -694.248,Z 969.467,A 0.000,B 0.000,C 90.000,E1 120.050} C_DIS
LIN {X -0.053,Y -695.627,Z 969.463,A 0.000,B 0.000,C 90.000,E1 119.333} C_DIS
LIN {X 0.353,Y -696.924,Z 969.458,A 0.000,B 0.000,C 90.000,E1 118.359} C_DIS
LIN {X 0.100,Y -698.159,Z 969.451,A 0.000,B 0.000,C 90.000,E1 117.206} C_DIS
LIN {X -0.087,Y -698.963,Z 969.446,A 0.000,B 0.000,C 90.000,E1 116.283} C_DIS
LIN {X 0.047,Y -699.555,Z 969.441,A 0.000,B 0.000,C 90.000,E1 115.335} C_DIS
LIN {X -0.078,Y -699.779,Z 969.437,A 0.000,B 0.000,C 90.000,E1 114.643} C_DIS
LIN {X 0.170,Y -699.738,Z 969.434,A 0.000,B 0.000,C 90.000,E1 114.155} C_DIS
LIN {X 0.066,Y -699.392,Z 969.432,A 0.000,B 0.000,C 90.000,E1 113.695} C_DIS
LIN {X 0.315,Y -698.097,Z 969.429,A 0.000,B 0.000,C 90.000,E1 113.206} C_DIS
LIN {X -0.066,Y -697.323,Z 969.428,A 0.000,B 0.000,C 90.000,E1 113.003} C_DIS
LIN {X -0.209,Y -696.627,Z 969.427,A 0.000,B 0.000,C 90.000,E1 112.898} C_DIS
LIN {X 0.029,Y -692.751,Z 969.425,A 0.000,B 0.000,C 90.000,E1 112.408} C_DIS
LIN {X 0.151,Y -691.541,Z 969.424,A 0.000,B 0.000,C 90.000,E1 112.280} C_DIS
LIN {X 0.289,Y -689.680,Z 969.423,A 0.000,B 0.000,C 90.000,E1 112.153} C_DIS
LIN {X 0.233,Y -685.238,Z 969.422,A 0.000,B 0.000,C 90.000,E1 111.972} C_DIS
LIN {X 0.262,Y -681.186,Z 969.422,A 0.000,B 0.000,C 90.000,E1 111.844} C_DIS
LIN {X -0.093,Y -677.117,Z 969.421,A 0.000,B 0.000,C 90.000,E1 111.770} C_DIS
LIN {X -0.033,Y -674.082,Z 969.421,A 0.000,B 0.000,C 90.000,E1 111.716} C_DIS
LIN {X -0.279,Y -667.202,Z 969.421,A 0.000,B 0.000,C 90.000,E1 111.716} C_DIS
LIN {X -0.299,Y -626.890,Z 969.421,A 0.000,B 0.000,C 90.000,E1 111.716} C_DIS
LIN {X 0.113,Y -621.589,Z 969.420,A 0.000,B 0.000,C 90.000,E1 111.589} C_DIS
LIN {X 0.054,Y -615.841,Z 969.419,A 0.000,B 0.000,C 90.000,E1 111.461} C_DIS
LIN {X 0.101,Y -608.901,Z 969.418,A 0.000,B 0.000,C 90.000,E1 111.227} C_DIS
LIN {X 0.033,Y -604.431,Z 969.417,A 0.000,B 0.000,C 90.000,E1 111.046} C_DIS
LIN {X -0.366,Y -597.892,Z 969.415,A 0.000,B 0.000,C 90.000,E1 110.737} C_DIS
LIN {X -0.152,Y -590.672,Z 969.412,A 0.000,B 0.000,C 90.000,E1 110.248} C_DIS
LIN {X 0.008,Y -576.356,Z 969.406,A 0.000,B 0.000,C 90.000,E1 109.141} C_DIS
LIN {X -0.022,Y -574.855,Z 969.406,A 0.000,B 0.000,C 90.000,E1 109.033} C_DIS
LIN {X -0.026,Y -566.533,Z 969.403,A 0.000,B 0.000,C 90.000,E1 108.544} C_DIS
LIN {X 0.124,Y -552.514,Z 969.399,A 0.000,B 0.000,C 90.000,E1 107.819} C_DIS
LIN {X -0.041,Y -550.303,Z 969.398,A 0.000,B 0.000,C 90.000,E1 107.638} C_DIS
LIN {X -0.079,Y -550.266,Z 969.398,A 0.000,B 0.000,C 90.000,E1 107.638} C_DIS
